LIN {X 0,Y 474.609,Z 227.864,A -85,B 0,C 180,E1 -7320.228,E2 -7320.228} C_VEL
LIN {X 0,Y 474.64,Z 227.86,A -85,B 0,C 180,E1 -7323.218,E2 -7323.218} C_VEL
LIN {X 0,Y 474.588,Z 227.869,A -85,B 0,C 180,E1 -7326.321,E2 -7326.321} C_VEL
LIN {X 0,Y 474.625,Z 227.862,A -85,B 0,C 180,E1 -7329.545,E2 -7329.545} C_VEL
LIN {X 0,Y 474.587,Z 227.87,A -85,B 0,C 180,E1 -7332.228,E2 -7332.228} C_VEL
LIN {X 0,Y 474.618,Z 227.86,A -85,B 0,C 180,E1 -7335.295,E2 -7335.295} C_VEL
LIN {X 0,Y 474.594,Z 227.868,A -85,B 0,C 180,E1 -7338.208,E2 -7338.208} C_VEL
LIN {X 0,Y 474.619,Z 227.864,A -85,B 0,C 180,E1 -7340.448,E2 -7340.448} C_VEL
LIN {X 0,Y 474.57,Z 227.865,A -85,B 0,C 180,E1 -7343.671,E2 -7343.671} C_VEL
LIN {X 0,Y 474.614,Z 227.864,A -85,B 0,C 180,E1 -7346.774,E2 -7346.774} C_VEL
LIN {X 0,Y 474.592,Z 227.863,A -85,B 0,C 180,E1 -7349.765,E2 -7349.765} C_VEL
LIN {X 0,Y 474.599,Z 227.867,A -85,B 0,C 180,E1 -7352.68,E2 -7352.68} C_VEL
LIN {X 0,Y 474.619,Z 227.86,A -85,B 0,C 180,E1 -7355.501,E2 -7355.501} C_VEL
LIN {X 0,Y 474.642,Z 227.86,A -85,B 0,C 180,E1 -7359.18,E2 -7359.18} C_VEL
LIN {X 0,Y 474.606,Z 227.861,A -85,B 0,C 180,E1 -7361.878,E2 -7361.878} C_VEL
LIN {X 0,Y 474.671,Z 227.856,A -85,B 0,C 180,E1 -7364.539,E2 -7364.539} C_VEL
LIN {X 0,Y 474.692,Z 227.848,A -85,B 0,C 180,E1 -7368.032,E2 -7368.032} C_VEL
LIN {X 0,Y 474.682,Z 227.855,A -85,B 0,C 180,E1 -7371.481,E2 -7371.481} C_VEL
LIN {X 0,Y 474.742,Z 227.843,A -85,B 0,C 180,E1 -7374.047,E2 -7374.047} C_VEL
LIN {X 0,Y 474.862,Z 227.835,A -85,B 0,C 180,E1 -7377.45,E2 -7377.45} C_VEL
LIN {X 0,Y 474.888,Z 227.826,A -85,B 0,C 180,E1 -7379.994,E2 -7379.994} C_VEL
LIN {X 0,Y 474.871,Z 227.828,A -85,B 0,C 180,E1 -7382.539,E2 -7382.539} C_VEL
LIN {X 0,Y 474.738,Z 227.848,A -85,B 0,C 180,E1 -7385.942,E2 -7385.942} C_VEL
LIN {X 0,Y 474.703,Z 227.851,A -85,B 0,C 180,E1 -7388.508,E2 -7388.508} C_VEL
LIN {X 0,Y 474.711,Z 227.853,A -85,B 0,C 180,E1 -7391.956,E2 -7391.956} C_VEL
LIN {X 0,Y 474.67,Z 227.86,A -85,B 0,C 180,E1 -7395.45,E2 -7395.45} C_VEL
LIN {X 0,Y 474.631,Z 227.862,A -85,B 0,C 180,E1 -7399.004,E2 -7399.004} C_VEL
LIN {X 0,Y 474.608,Z 227.868,A -85,B 0,C 180,E1 -7401.72,E2 -7401.72} C_VEL
LIN {X 0,Y 474.67,Z 227.981,A -85,B 0,C 180,E1 -7403.845,E2 -7403.845} C_VEL
LIN {X 0,Y 475.847,Z 234.41,A -85,B 0,C 180,E1 -7405.119,E2 -7405.119} C_VEL
LIN {X 0,Y 475.431,Z 251.659,A -85,B 0,C 180,E1 -7408.223,E2 -7408.223} C_VEL
LIN {X 0,Y 475.369,Z 257.615,A -85,B 0,C 180,E1 -7409.254,E2 -7409.254} C_VEL
LIN {X 0,Y 478.155,Z 273.903,A -85,B 0,C 180,E1 -7409.639,E2 -7409.639} C_VEL
LIN {X 0,Y 477.321,Z 365.648,A -85,B 0,C 180,E1 -7411.09,E2 -7411.09} C_VEL
LIN {X 0,Y 477,Z 379.548,A -85,B 0,C 180,E1 -7411.494,E2 -7411.494} C_VEL
LIN {X 0,Y 476.715,Z 392.201,A -85,B 0,C 180,E1 -7412.046,E2 -7412.046} C_VEL
LIN {X 0,Y 476.272,Z 404.083,A -85,B 0,C 180,E1 -7412.747,E2 -7412.747} C_VEL
LIN {X 0,Y 475.72,Z 415.798,A -85,B 0,C 180,E1 -7413.633,E2 -7413.633} C_VEL
LIN {X 0,Y 475.327,Z 425.567,A -85,B 0,C 180,E1 -7414.559,E2 -7414.559} C_VEL
LIN {X 0,Y 474.857,Z 435.029,A -85,B 0,C 180,E1 -7415.666,E2 -7415.666} C_VEL
LIN {X 0,Y 474.48,Z 443.518,A -85,B 0,C 180,E1 -7416.888,E2 -7416.888} C_VEL
LIN {X 0,Y 474.188,Z 451.047,A -85,B 0,C 180,E1 -7418.235,E2 -7418.235} C_VEL
LIN {X 0,Y 473.959,Z 457.052,A -85,B 0,C 180,E1 -7419.604,E2 -7419.604} C_VEL
LIN {X 0,Y 473.835,Z 461.346,A -85,B 0,C 180,E1 -7420.852,E2 -7420.852} C_VEL
LIN {X 0,Y 473.699,Z 464.658,A -85,B 0,C 180,E1 -7422.116,E2 -7422.116} C_VEL
LIN {X 0,Y 473.616,Z 466.97,A -85,B 0,C 180,E1 -7423.358,E2 -7423.358} C_VEL
LIN {X 0,Y 473.635,Z 468.364,A -85,B 0,C 180,E1 -7424.585,E2 -7424.585} C_VEL
LIN {X 0,Y 473.606,Z 468.909,A -85,B 0,C 180,E1 -7425.78,E2 -7425.78} C_VEL
LIN {X 0,Y 473.574,Z 468.694,A -85,B 0,C 180,E1 -7426.951,E2 -7426.951} C_VEL
LIN {X 0,Y 473.665,Z 467.748,A -85,B 0,C 180,E1 -7428.114,E2 -7428.114} C_VEL
LIN {X 0,Y 473.705,Z 464.944,A -85,B 0,C 180,E1 -7429.809,E2 -7429.809} C_VEL
LIN {X 0,Y 473.85,Z 460.634,A -85,B 0,C 180,E1 -7431.445,E2 -7431.445} C_VEL
LIN {X 0,Y 473.285,Z 458.514,A -85,B 0,C 180,E1 -7432.109,E2 -7432.109} C_VEL
LIN {X 0,Y 470.568,Z 454.555,A -85,B 0,C 180,E1 -7433.163,E2 -7433.163} C_VEL
LIN {X 0,Y 467.86,Z 449.885,A -85,B 0,C 180,E1 -7434.184,E2 -7434.184} C_VEL
LIN {X 0,Y 467.32,Z 446.646,A -85,B 0,C 180,E1 -7434.789,E2 -7434.789} C_VEL
LIN {X 0,Y 467.621,Z 439.191,A -85,B 0,C 180,E1 -7435.983,E2 -7435.983} C_VEL
LIN {X 0,Y 468.08,Z 429.769,A -85,B 0,C 180,E1 -7437.209,E2 -7437.209} C_VEL
LIN {X 0,Y 468.529,Z 420.264,A -85,B 0,C 180,E1 -7438.207,E2 -7438.207} C_VEL
LIN {X 0,Y 469.018,Z 409.141,A -85,B 0,C 180,E1 -7439.149,E2 -7439.149} C_VEL
LIN {X 0,Y 469.526,Z 397.344,A -85,B 0,C 180,E1 -7439.938,E2 -7439.938} C_VEL
LIN {X 0,Y 469.937,Z 385.154,A -85,B 0,C 180,E1 -7440.553,E2 -7440.553} C_VEL
LIN {X 0,Y 470.285,Z 372.084,A -85,B 0,C 180,E1 -7441.021,E2 -7441.021} C_VEL
LIN {X 0,Y 470.513,Z 359.082,A -85,B 0,C 180,E1 -7441.311,E2 -7441.311} C_VEL
LIN {X 0,Y 471.128,Z 273.425,A -85,B 0,C 180,E1 -7442.668,E2 -7442.668} C_VEL
LIN {X 0,Y 468.516,Z 258.548,A -85,B 0,C 180,E1 -7443.016,E2 -7443.016} C_VEL
LIN {X 0,Y 468.469,Z 257.54,A -85,B 0,C 180,E1 -7443.134,E2 -7443.134} C_VEL
LIN {X 0,Y 469.141,Z 241.607,A -85,B 0,C 180,E1 -7446.378,E2 -7446.378} C_VEL
LIN {X 0,Y 469.154,Z 237.141,A -85,B 0,C 180,E1 -7447.312,E2 -7447.312} C_VEL
LIN {X 0,Y 467.581,Z 228.795,A -85,B 0,C 180,E1 -7449.203,E2 -7449.203} C_VEL
LIN {X 0,Y 467.534,Z 228.751,A -85,B 0,C 180,E1 -7452.506,E2 -7452.506} C_VEL
LIN {X 0,Y 467.55,Z 228.741,A -85,B 0,C 180,E1 -7455.196,E2 -7455.196} C_VEL
LIN {X 0,Y 467.62,Z 228.731,A -85,B 0,C 180,E1 -7457.855,E2 -7457.855} C_VEL
LIN {X 0,Y 467.611,Z 228.733,A -85,B 0,C 180,E1 -7461.358,E2 -7461.358} C_VEL
LIN {X 0,Y 467.677,Z 228.724,A -85,B 0,C 180,E1 -7463.963,E2 -7463.963} C_VEL
LIN {X 0,Y 467.792,Z 228.712,A -85,B 0,C 180,E1 -7467.418,E2 -7467.418} C_VEL
LIN {X 0,Y 467.802,Z 228.708,A -85,B 0,C 180,E1 -7470.001,E2 -7470.001} C_VEL
LIN {X 0,Y 467.793,Z 228.711,A -85,B 0,C 180,E1 -7472.585,E2 -7472.585} C_VEL
LIN {X 0,Y 467.679,Z 228.724,A -85,B 0,C 180,E1 -7476.04,E2 -7476.04} C_VEL
LIN {X 0,Y 467.615,Z 228.732,A -85,B 0,C 180,E1 -7478.645,E2 -7478.645} C_VEL
LIN {X 0,Y 467.625,Z 228.731,A -85,B 0,C 180,E1 -7482.148,E2 -7482.148} C_VEL
LIN {X 0,Y 467.57,Z 228.744,A -85,B 0,C 180,E1 -7485.699,E2 -7485.699} C_VEL
LIN {X 0,Y 467.547,Z 228.74,A -85,B 0,C 180,E1 -7488.768,E2 -7488.768} C_VEL
LIN {X 0,Y 467.514,Z 228.747,A -85,B 0,C 180,E1 -7491.273,E2 -7491.273} C_VEL
LIN {X 0,Y 467.511,Z 228.751,A -85,B 0,C 180,E1 -7493.948,E2 -7493.948} C_VEL
LIN {X 0,Y 467.565,Z 228.738,A -85,B 0,C 180,E1 -7496.805,E2 -7496.805} C_VEL
LIN {X 0,Y 467.529,Z 228.747,A -85,B 0,C 180,E1 -7499.741,E2 -7499.741} C_VEL
LIN {X 0,Y 467.527,Z 228.743,A -85,B 0,C 180,E1 -7502.764,E2 -7502.764} C_VEL
LIN {X 0,Y 467.502,Z 228.75,A -85,B 0,C 180,E1 -7505.895,E2 -7505.895} C_VEL
LIN {X 0,Y 467.549,Z 228.74,A -85,B 0,C 180,E1 -7509.149,E2 -7509.149} C_VEL
LIN {X 0,Y 467.573,Z 228.744,A -85,B 0,C 180,E1 -7512.578,E2 -7512.578} C_VEL
LIN {X 0,Y 467.534,Z 228.746,A -85,B 0,C 180,E1 -7516.265,E2 -7516.265} C_VEL
LIN {X 0,Y 467.551,Z 228.747,A -85,B 0,C 180,E1 -7518.728,E2 -7518.728} C_VEL
LIN {X 0,Y 467.54,Z 228.742,A -85,B 0,C 180,E1 -7521.414,E2 -7521.414} C_VEL
LIN {X 0,Y 467.529,Z 228.744,A -85,B 0,C 180,E1 -7524.268,E2 -7524.268} C_VEL
LIN {X 0,Y 467.551,Z 228.743,A -85,B 0,C 180,E1 -7527.328,E2 -7527.328} C_VEL
LIN {X 0,Y 467.544,Z 228.744,A -85,B 0,C 180,E1 -7530.675,E2 -7530.675} C_VEL
LIN {X 0,Y 467.594,Z 228.742,A -85,B 0,C 180,E1 -7533.207,E2 -7533.207} C_VEL
LIN {X 0,Y 467.574,Z 228.737,A -85,B 0,C 180,E1 -7536.475,E2 -7536.475} C_VEL
LIN {X 0,Y 467.608,Z 228.735,A -85,B 0,C 180,E1 -7539.784,E2 -7539.784} C_VEL
LIN {X 0,Y 467.586,Z 228.735,A -85,B 0,C 180,E1 -7542.513,E2 -7542.513} C_VEL
LIN {X 0,Y 467.596,Z 228.737,A -85,B 0,C 180,E1 -7545.203,E2 -7545.203} C_VEL
LIN {X 0,Y 467.65,Z 228.733,A -85,B 0,C 180,E1 -7547.861,E2 -7547.861} C_VEL
LIN {X 0,Y 467.667,Z 228.728,A -85,B 0,C 180,E1 -7551.363,E2 -7551.363} C_VEL
LIN {X 0,Y 467.712,Z 228.727,A -85,B 0,C 180,E1 -7553.968,E2 -7553.968} C_VEL
LIN {X 0,Y 467.851,Z 228.704,A -85,B 0,C 180,E1 -7557.423,E2 -7557.423} C_VEL
LIN {X 0,Y 467.854,Z 228.71,A -85,B 0,C 180,E1 -7560.006,E2 -7560.006} C_VEL
LIN {X 0,Y 467.819,Z 228.709,A -85,B 0,C 180,E1 -7562.589,E2 -7562.589} C_VEL
LIN {X 0,Y 467.714,Z 228.725,A -85,B 0,C 180,E1 -7566.043,E2 -7566.043} C_VEL
LIN {X 0,Y 467.646,Z 228.732,A -85,B 0,C 180,E1 -7568.649,E2 -7568.649} C_VEL
LIN {X 0,Y 467.669,Z 228.729,A -85,B 0,C 180,E1 -7572.15,E2 -7572.15} C_VEL
LIN {X 0,Y 467.664,Z 228.726,A -85,B 0,C 180,E1 -7575.889,E2 -7575.889} C_VEL
LIN {X 0,Y 467.636,Z 228.73,A -85,B 0,C 180,E1 -7579.312,E2 -7579.312} C_VEL
LIN {X 0,Y 467.548,Z 228.74,A -85,B 0,C 180,E1 -7582.078,E2 -7582.078} C_VEL
LIN {X 0,Y 467.574,Z 228.746,A -85,B 0,C 180,E1 -7584.893,E2 -7584.893} C_VEL
LIN {X 0,Y 467.564,Z 228.738,A -85,B 0,C 180,E1 -7587.777,E2 -7587.777} C_VEL
LIN {X 0,Y 467.566,Z 228.745,A -85,B 0,C 180,E1 -7591.043,E2 -7591.043} C_VEL
LIN {X 0,Y 467.595,Z 228.734,A -85,B 0,C 180,E1 -7594.242,E2 -7594.242} C_VEL
LIN {X 0,Y 467.561,Z 228.745,A -85,B 0,C 180,E1 -7597.187,E2 -7597.187} C_VEL
LIN {X 0,Y 467.577,Z 228.736,A -85,B 0,C 180,E1 -7600.269,E2 -7600.269} C_VEL
LIN {X 0,Y 467.537,Z 228.741,A -85,B 0,C 180,E1 -7602.57,E2 -7602.57} C_VEL
LIN {X 0,Y 467.574,Z 228.738,A -85,B 0,C 180,E1 -7605.052,E2 -7605.052} C_VEL
LIN {X 0,Y 467.58,Z 228.736,A -85,B 0,C 180,E1 -7608.727,E2 -7608.727} C_VEL
LIN {X 0,Y 467.562,Z 228.745,A -85,B 0,C 180,E1 -7611.954,E2 -7611.954} C_VEL
LIN {X 0,Y 467.573,Z 228.737,A -85,B 0,C 180,E1 -7615.167,E2 -7615.167} C_VEL
LIN {X 0,Y 467.596,Z 228.742,A -85,B 0,C 180,E1 -7618.26,E2 -7618.26} C_VEL
LIN {X 0,Y 467.573,Z 228.74,A -85,B 0,C 180,E1 -7621.249,E2 -7621.249} C_VEL
LIN {X 0,Y 467.6,Z 228.742,A -85,B 0,C 180,E1 -7624.158,E2 -7624.158} C_VEL
LIN {X 0,Y 467.637,Z 228.864,A -85,B 0,C 180,E1 -7625.061,E2 -7625.061} C_VEL
LIN {X 0,Y 469.628,Z 239.857,A -85,B 0,C 180,E1 -7627.333,E2 -7627.333} C_VEL
LIN {X 0,Y 469.11,Z 253.106,A -85,B 0,C 180,E1 -7629.843,E2 -7629.843} C_VEL
LIN {X 0,Y 468.404,Z 270.161,A -85,B 0,C 180,E1 -7632.986,E2 -7632.986} C_VEL
LIN {X 0,Y 469.313,Z 275.962,A -85,B 0,C 180,E1 -7633.15,E2 -7633.15} C_VEL
LIN {X 0,Y 471.214,Z 288.215,A -85,B 0,C 180,E1 -7633.414,E2 -7633.414} C_VEL
LIN {X 0,Y 470.431,Z 377.814,A -85,B 0,C 180,E1 -7634.843,E2 -7634.843} C_VEL
LIN {X 0,Y 470.097,Z 391.028,A -85,B 0,C 180,E1 -7635.22,E2 -7635.22} C_VEL
LIN {X 0,Y 469.668,Z 403.753,A -85,B 0,C 180,E1 -7635.76,E2 -7635.76} C_VEL
LIN {X 0,Y 469.197,Z 415.879,A -85,B 0,C 180,E1 -7636.463,E2 -7636.463} C_VEL
LIN {X 0,Y 468.757,Z 426.287,A -85,B 0,C 180,E1 -7637.236,E2 -7637.236} C_VEL
LIN {X 0,Y 468.268,Z 436.753,A -85,B 0,C 180,E1 -7638.199,E2 -7638.199} C_VEL
LIN {X 0,Y 467.808,Z 445.435,A -85,B 0,C 180,E1 -7639.175,E2 -7639.175} C_VEL
LIN {X 0,Y 467.479,Z 453.433,A -85,B 0,C 180,E1 -7640.261,E2 -7640.261} C_VEL
LIN {X 0,Y 467.157,Z 461.253,A -85,B 0,C 180,E1 -7641.564,E2 -7641.564} C_VEL
LIN {X 0,Y 466.862,Z 468.418,A -85,B 0,C 180,E1 -7643.082,E2 -7643.082} C_VEL
LIN {X 0,Y 466.795,Z 473.191,A -85,B 0,C 180,E1 -7644.382,E2 -7644.382} C_VEL
LIN {X 0,Y 466.651,Z 476.837,A -85,B 0,C 180,E1 -7645.68,E2 -7645.68} C_VEL
LIN {X 0,Y 466.665,Z 478.72,A -85,B 0,C 180,E1 -7646.545,E2 -7646.545} C_VEL
LIN {X 0,Y 466.648,Z 480.133,A -85,B 0,C 180,E1 -7647.409,E2 -7647.409} C_VEL
LIN {X 0,Y 466.593,Z 481.751,A -85,B 0,C 180,E1 -7649.135,E2 -7649.135} C_VEL
LIN {X 0,Y 466.603,Z 481.973,A -85,B 0,C 180,E1 -7649.999,E2 -7649.999} C_VEL
LIN {X 0,Y 466.593,Z 481.757,A -85,B 0,C 180,E1 -7650.862,E2 -7650.862} C_VEL
LIN {X 0,Y 466.648,Z 480.142,A -85,B 0,C 180,E1 -7652.588,E2 -7652.588} C_VEL
LIN {X 0,Y 466.664,Z 478.736,A -85,B 0,C 180,E1 -7653.452,E2 -7653.452} C_VEL
LIN {X 0,Y 466.694,Z 475.781,A -85,B 0,C 180,E1 -7654.749,E2 -7654.749} C_VEL
LIN {X 0,Y 466.779,Z 471.78,A -85,B 0,C 180,E1 -7656.048,E2 -7656.048} C_VEL
LIN {X 0,Y 466.983,Z 465.623,A -85,B 0,C 180,E1 -7657.565,E2 -7657.565} C_VEL
LIN {X 0,Y 467.274,Z 458.899,A -85,B 0,C 180,E1 -7658.867,E2 -7658.867} C_VEL
LIN {X 0,Y 467.616,Z 450.554,A -85,B 0,C 180,E1 -7660.17,E2 -7660.17} C_VEL
LIN {X 0,Y 468.03,Z 441.975,A -85,B 0,C 180,E1 -7661.255,E2 -7661.255} C_VEL
LIN {X 0,Y 468.555,Z 431.775,A -85,B 0,C 180,E1 -7662.304,E2 -7662.304} C_VEL
LIN {X 0,Y 468.977,Z 420.901,A -85,B 0,C 180,E1 -7663.209,E2 -7663.209} C_VEL
LIN {X 0,Y 469.468,Z 409.359,A -85,B 0,C 180,E1 -7663.967,E2 -7663.967} C_VEL
LIN {X 0,Y 469.935,Z 397.4,A -85,B 0,C 180,E1 -7664.561,E2 -7664.561} C_VEL
LIN {X 0,Y 470.353,Z 383.614,A -85,B 0,C 180,E1 -7665.046,E2 -7665.046} C_VEL
LIN {X 0,Y 470.587,Z 370.995,A -85,B 0,C 180,E1 -7665.315,E2 -7665.315} C_VEL
LIN {X 0,Y 471.217,Z 286.858,A -85,B 0,C 180,E1 -7666.654,E2 -7666.654} C_VEL
LIN {X 0,Y 468.38,Z 269.763,A -85,B 0,C 180,E1 -7667.072,E2 -7667.072} C_VEL
LIN {X 0,Y 468.952,Z 253.914,A -85,B 0,C 180,E1 -7669.933,E2 -7669.933} C_VEL
LIN {X 0,Y 469.534,Z 240.329,A -85,B 0,C 180,E1 -7672.436,E2 -7672.436} C_VEL
LIN {X 0,Y 468.428,Z 232.889,A -85,B 0,C 180,E1 -7673.895,E2 -7673.895} C_VEL
LIN {X 0,Y 467.616,Z 228.82,A -85,B 0,C 180,E1 -7674.766,E2 -7674.766} C_VEL
LIN {X 0,Y 467.623,Z 228.738,A -85,B 0,C 180,E1 -7677.767,E2 -7677.767} C_VEL
LIN {X 0,Y 467.573,Z 228.738,A -85,B 0,C 180,E1 -7681.041,E2 -7681.041} C_VEL
LIN {X 0,Y 467.594,Z 228.74,A -85,B 0,C 180,E1 -7684.239,E2 -7684.239} C_VEL
LIN {X 0,Y 467.546,Z 228.743,A -85,B 0,C 180,E1 -7687.182,E2 -7687.182} C_VEL
LIN {X 0,Y 467.562,Z 228.745,A -85,B 0,C 180,E1 -7690.264,E2 -7690.264} C_VEL
LIN {X 0,Y 467.549,Z 228.743,A -85,B 0,C 180,E1 -7693.742,E2 -7693.742} C_VEL
LIN {X 0,Y 467.547,Z 228.748,A -85,B 0,C 180,E1 -7696.251,E2 -7696.251} C_VEL
LIN {X 0,Y 467.558,Z 228.742,A -85,B 0,C 180,E1 -7699.729,E2 -7699.729} C_VEL
LIN {X 0,Y 467.516,Z 228.746,A -85,B 0,C 180,E1 -7702.815,E2 -7702.815} C_VEL
LIN {X 0,Y 467.575,Z 228.739,A -85,B 0,C 180,E1 -7705.756,E2 -7705.756} C_VEL
LIN {X 0,Y 467.545,Z 228.743,A -85,B 0,C 180,E1 -7708.956,E2 -7708.956} C_VEL
LIN {X 0,Y 467.541,Z 228.746,A -85,B 0,C 180,E1 -7712.222,E2 -7712.222} C_VEL
LIN {X 0,Y 467.551,Z 228.744,A -85,B 0,C 180,E1 -7715.105,E2 -7715.105} C_VEL
LIN {X 0,Y 467.517,Z 228.743,A -85,B 0,C 180,E1 -7717.921,E2 -7717.921} C_VEL
LIN {X 0,Y 467.546,Z 228.745,A -85,B 0,C 180,E1 -7720.684,E2 -7720.684} C_VEL
LIN {X 0,Y 467.585,Z 228.735,A -85,B 0,C 180,E1 -7724.135,E2 -7724.135} C_VEL
LIN {X 0,Y 467.643,Z 228.727,A -85,B 0,C 180,E1 -7727.638,E2 -7727.638} C_VEL
LIN {X 0,Y 467.642,Z 228.733,A -85,B 0,C 180,E1 -7731.351,E2 -7731.351} C_VEL
LIN {X 0,Y 467.707,Z 228.719,A -85,B 0,C 180,E1 -7733.957,E2 -7733.957} C_VEL
LIN {X 0,Y 467.803,Z 228.714,A -85,B 0,C 180,E1 -7737.411,E2 -7737.411} C_VEL
LIN {X 0,Y 467.859,Z 228.701,A -85,B 0,C 180,E1 -7739.994,E2 -7739.994} C_VEL
LIN {X 0,Y 467.837,Z 228.705,A -85,B 0,C 180,E1 -7742.577,E2 -7742.577} C_VEL
LIN {X 0,Y 467.7,Z 228.724,A -85,B 0,C 180,E1 -7746.032,E2 -7746.032} C_VEL
LIN {X 0,Y 467.657,Z 228.729,A -85,B 0,C 180,E1 -7748.637,E2 -7748.637} C_VEL
LIN {X 0,Y 467.663,Z 228.728,A -85,B 0,C 180,E1 -7752.373,E2 -7752.373} C_VEL
LIN {X 0,Y 467.618,Z 228.739,A -85,B 0,C 180,E1 -7755.88,E2 -7755.88} C_VEL
LIN {X 0,Y 467.59,Z 228.741,A -85,B 0,C 180,E1 -7759.302,E2 -7759.302} C_VEL
LIN {X 0,Y 467.543,Z 228.748,A -85,B 0,C 180,E1 -7762.066,E2 -7762.066} C_VEL
LIN {X 0,Y 467.633,Z 228.785,A -85,B 0,C 180,E1 -7763.61,E2 -7763.61} C_VEL
LIN {X 0,Y 468.567,Z 233.439,A -85,B 0,C 180,E1 -7764.588,E2 -7764.588} C_VEL
LIN {X 0,Y 468.961,Z 237.071,A -85,B 0,C 180,E1 -7765.276,E2 -7765.276} C_VEL
LIN {X 0,Y 468.449,Z 254.311,A -85,B 0,C 180,E1 -7768.413,E2 -7768.413} C_VEL
LIN {X 0,Y 468.408,Z 257.7,A -85,B 0,C 180,E1 -7768.985,E2 -7768.985} C_VEL
LIN {X 0,Y 471.352,Z 273.713,A -85,B 0,C 180,E1 -7769.382,E2 -7769.382} C_VEL
LIN {X 0,Y 470.48,Z 366.047,A -85,B 0,C 180,E1 -7770.872,E2 -7770.872} C_VEL
LIN {X 0,Y 470.127,Z 380.038,A -85,B 0,C 180,E1 -7771.289,E2 -7771.289} C_VEL
LIN {X 0,Y 469.829,Z 391.909,A -85,B 0,C 180,E1 -7771.813,E2 -7771.813} C_VEL
LIN {X 0,Y 469.359,Z 403.284,A -85,B 0,C 180,E1 -7772.482,E2 -7772.482} C_VEL
LIN {X 0,Y 468.822,Z 415.254,A -85,B 0,C 180,E1 -7773.39,E2 -7773.39} C_VEL
LIN {X 0,Y 468.349,Z 425.658,A -85,B 0,C 180,E1 -7774.382,E2 -7774.382} C_VEL
LIN {X 0,Y 467.838,Z 435.416,A -85,B 0,C 180,E1 -7775.544,E2 -7775.544} C_VEL
LIN {X 0,Y 467.468,Z 443.261,A -85,B 0,C 180,E1 -7776.689,E2 -7776.689} C_VEL
LIN {X 0,Y 467.138,Z 450.965,A -85,B 0,C 180,E1 -7778.075,E2 -7778.075} C_VEL
LIN {X 0,Y 466.883,Z 457.229,A -85,B 0,C 180,E1 -7779.523,E2 -7779.523} C_VEL
LIN {X 0,Y 466.728,Z 462.57,A -85,B 0,C 180,E1 -7781.161,E2 -7781.161} C_VEL
LIN {X 0,Y 466.579,Z 465.989,A -85,B 0,C 180,E1 -7782.663,E2 -7782.663} C_VEL
LIN {X 0,Y 466.535,Z 467.769,A -85,B 0,C 180,E1 -7783.853,E2 -7783.853} C_VEL
LIN {X 0,Y 466.532,Z 468.774,A -85,B 0,C 180,E1 -7785.062,E2 -7785.062} C_VEL
LIN {X 0,Y 466.475,Z 469.004,A -85,B 0,C 180,E1 -7786.305,E2 -7786.305} C_VEL
LIN {X 0,Y 466.508,Z 468.399,A -85,B 0,C 180,E1 -7787.565,E2 -7787.565} C_VEL
LIN {X 0,Y 466.569,Z 466.896,A -85,B 0,C 180,E1 -7788.851,E2 -7788.851} C_VEL
LIN {X 0,Y 466.628,Z 464.383,A -85,B 0,C 180,E1 -7790.172,E2 -7790.172} C_VEL
LIN {X 0,Y 466.774,Z 460.754,A -85,B 0,C 180,E1 -7791.516,E2 -7791.516} C_VEL
LIN {X 0,Y 466.963,Z 455.403,A -85,B 0,C 180,E1 -7792.988,E2 -7792.988} C_VEL
LIN {X 0,Y 467.205,Z 449.264,A -85,B 0,C 180,E1 -7794.306,E2 -7794.306} C_VEL
LIN {X 0,Y 467.32,Z 446.646,A -85,B 0,C 180,E1 -7794.789,E2 -7794.789} C_VEL
LIN {X 0,Y 466.807,Z 443.26,A -85,B 0,C 180,E1 -7795.377,E2 -7795.377} C_VEL
LIN {X 0,Y 464.234,Z 437.436,A -85,B 0,C 180,E1 -7796.313,E2 -7796.313} C_VEL
LIN {X 0,Y 461.697,Z 431.084,A -85,B 0,C 180,E1 -7797.202,E2 -7797.202} C_VEL
LIN {X 0,Y 461.245,Z 426.806,A -85,B 0,C 180,E1 -7797.712,E2 -7797.712} C_VEL
LIN {X 0,Y 461.776,Z 416.304,A -85,B 0,C 180,E1 -7798.755,E2 -7798.755} C_VEL
LIN {X 0,Y 462.293,Z 405.076,A -85,B 0,C 180,E1 -7799.639,E2 -7799.639} C_VEL
LIN {X 0,Y 462.766,Z 393.347,A -85,B 0,C 180,E1 -7800.364,E2 -7800.364} C_VEL
LIN {X 0,Y 463.168,Z 380.581,A -85,B 0,C 180,E1 -7800.953,E2 -7800.953} C_VEL
LIN {X 0,Y 463.522,Z 367.51,A -85,B 0,C 180,E1 -7801.358,E2 -7801.358} C_VEL
LIN {X 0,Y 463.75,Z 344.948,A -85,B 0,C 180,E1 -7801.755,E2 -7801.755} C_VEL
LIN {X 0,Y 464.275,Z 273.94,A -85,B 0,C 180,E1 -7802.902,E2 -7802.902} C_VEL
LIN {X 0,Y 461.546,Z 258.523,A -85,B 0,C 180,E1 -7803.279,E2 -7803.279} C_VEL
LIN {X 0,Y 461.528,Z 256.772,A -85,B 0,C 180,E1 -7803.553,E2 -7803.553} C_VEL
LIN {X 0,Y 462.19,Z 242.567,A -85,B 0,C 180,E1 -7806.502,E2 -7806.502} C_VEL
LIN {X 0,Y 462.17,Z 238.23,A -85,B 0,C 180,E1 -7807.422,E2 -7807.422} C_VEL
LIN {X 0,Y 460.515,Z 229.675,A -85,B 0,C 180,E1 -7809.395,E2 -7809.395} C_VEL
LIN {X 0,Y 460.483,Z 229.627,A -85,B 0,C 180,E1 -7812.229,E2 -7812.229} C_VEL
LIN {X 0,Y 460.51,Z 229.62,A -85,B 0,C 180,E1 -7814.965,E2 -7814.965} C_VEL
LIN {X 0,Y 460.6,Z 229.605,A -85,B 0,C 180,E1 -7817.667,E2 -7817.667} C_VEL
LIN {X 0,Y 460.558,Z 229.613,A -85,B 0,C 180,E1 -7821.224,E2 -7821.224} C_VEL
LIN {X 0,Y 460.641,Z 229.6,A -85,B 0,C 180,E1 -7823.871,E2 -7823.871} C_VEL
LIN {X 0,Y 460.758,Z 229.588,A -85,B 0,C 180,E1 -7827.379,E2 -7827.379} C_VEL
LIN {X 0,Y 460.774,Z 229.583,A -85,B 0,C 180,E1 -7830.001,E2 -7830.001} C_VEL
LIN {X 0,Y 460.759,Z 229.588,A -85,B 0,C 180,E1 -7832.624,E2 -7832.624} C_VEL
LIN {X 0,Y 460.643,Z 229.6,A -85,B 0,C 180,E1 -7836.132,E2 -7836.132} C_VEL
LIN {X 0,Y 460.561,Z 229.612,A -85,B 0,C 180,E1 -7838.779,E2 -7838.779} C_VEL
LIN {X 0,Y 460.562,Z 229.61,A -85,B 0,C 180,E1 -7842.46,E2 -7842.46} C_VEL
LIN {X 0,Y 460.53,Z 229.617,A -85,B 0,C 180,E1 -7846.001,E2 -7846.001} C_VEL
LIN {X 0,Y 460.501,Z 229.618,A -85,B 0,C 180,E1 -7848.905,E2 -7848.905} C_VEL
LIN {X 0,Y 460.449,Z 229.629,A -85,B 0,C 180,E1 -7851.49,E2 -7851.49} C_VEL
LIN {X 0,Y 460.483,Z 229.622,A -85,B 0,C 180,E1 -7854.337,E2 -7854.337} C_VEL
LIN {X 0,Y 460.522,Z 229.616,A -85,B 0,C 180,E1 -7857.248,E2 -7857.248} C_VEL
LIN {X 0,Y 460.47,Z 229.627,A -85,B 0,C 180,E1 -7860.244,E2 -7860.244} C_VEL
LIN {X 0,Y 460.473,Z 229.621,A -85,B 0,C 180,E1 -7863.331,E2 -7863.331} C_VEL
LIN {X 0,Y 460.425,Z 229.632,A -85,B 0,C 180,E1 -7866.535,E2 -7866.535} C_VEL
LIN {X 0,Y 460.525,Z 229.617,A -85,B 0,C 180,E1 -7869.864,E2 -7869.864} C_VEL
LIN {X 0,Y 460.496,Z 229.621,A -85,B 0,C 180,E1 -7872.911,E2 -7872.911} C_VEL
LIN {X 0,Y 460.481,Z 229.621,A -85,B 0,C 180,E1 -7875.836,E2 -7875.836} C_VEL
LIN {X 0,Y 460.505,Z 229.621,A -85,B 0,C 180,E1 -7878.997,E2 -7878.997} C_VEL
LIN {X 0,Y 460.509,Z 229.619,A -85,B 0,C 180,E1 -7881.276,E2 -7881.276} C_VEL
LIN {X 0,Y 460.479,Z 229.625,A -85,B 0,C 180,E1 -7884.562,E2 -7884.562} C_VEL
LIN {X 0,Y 460.502,Z 229.618,A -85,B 0,C 180,E1 -7887.723,E2 -7887.723} C_VEL
LIN {X 0,Y 460.514,Z 229.62,A -85,B 0,C 180,E1 -7890.776,E2 -7890.776} C_VEL
LIN {X 0,Y 460.538,Z 229.615,A -85,B 0,C 180,E1 -7893.742,E2 -7893.742} C_VEL
LIN {X 0,Y 460.528,Z 229.615,A -85,B 0,C 180,E1 -7896.631,E2 -7896.631} C_VEL
LIN {X 0,Y 460.537,Z 229.621,A -85,B 0,C 180,E1 -7899.46,E2 -7899.46} C_VEL
LIN {X 0,Y 460.537,Z 229.613,A -85,B 0,C 180,E1 -7902.237,E2 -7902.237} C_VEL
LIN {X 0,Y 460.555,Z 229.612,A -85,B 0,C 180,E1 -7904.972,E2 -7904.972} C_VEL
LIN {X 0,Y 460.604,Z 229.605,A -85,B 0,C 180,E1 -7908.566,E2 -7908.566} C_VEL
LIN {X 0,Y 460.617,Z 229.605,A -85,B 0,C 180,E1 -7911.23,E2 -7911.23} C_VEL
LIN {X 0,Y 460.678,Z 229.604,A -85,B 0,C 180,E1 -7913.876,E2 -7913.876} C_VEL
LIN {X 0,Y 460.791,Z 229.583,A -85,B 0,C 180,E1 -7917.383,E2 -7917.383} C_VEL
LIN {X 0,Y 460.823,Z 229.586,A -85,B 0,C 180,E1 -7920.006,E2 -7920.006} C_VEL
LIN {X 0,Y 460.763,Z 229.587,A -85,B 0,C 180,E1 -7922.628,E2 -7922.628} C_VEL
LIN {X 0,Y 460.679,Z 229.602,A -85,B 0,C 180,E1 -7926.136,E2 -7926.136} C_VEL
LIN {X 0,Y 460.602,Z 229.608,A -85,B 0,C 180,E1 -7928.782,E2 -7928.782} C_VEL
LIN {X 0,Y 460.623,Z 229.609,A -85,B 0,C 180,E1 -7932.339,E2 -7932.339} C_VEL
LIN {X 0,Y 460.617,Z 229.604,A -85,B 0,C 180,E1 -7936.002,E2 -7936.002} C_VEL
LIN {X 0,Y 460.582,Z 229.607,A -85,B 0,C 180,E1 -7939.62,E2 -7939.62} C_VEL
LIN {X 0,Y 460.525,Z 229.618,A -85,B 0,C 180,E1 -7942.433,E2 -7942.433} C_VEL
LIN {X 0,Y 460.551,Z 229.611,A -85,B 0,C 180,E1 -7945.796,E2 -7945.796} C_VEL
LIN {X 0,Y 460.539,Z 229.619,A -85,B 0,C 180,E1 -7949.235,E2 -7949.235} C_VEL
LIN {X 0,Y 460.537,Z 229.613,A -85,B 0,C 180,E1 -7952.288,E2 -7952.288} C_VEL
LIN {X 0,Y 460.524,Z 229.621,A -85,B 0,C 180,E1 -7955.449,E2 -7955.449} C_VEL
LIN {X 0,Y 460.523,Z 229.617,A -85,B 0,C 180,E1 -7958.893,E2 -7958.893} C_VEL
LIN {X 0,Y 460.522,Z 229.622,A -85,B 0,C 180,E1 -7961.6,E2 -7961.6} C_VEL
LIN {X 0,Y 460.517,Z 229.615,A -85,B 0,C 180,E1 -7964.593,E2 -7964.593} C_VEL
LIN {X 0,Y 460.493,Z 229.626,A -85,B 0,C 180,E1 -7967.814,E2 -7967.814} C_VEL
LIN {X 0,Y 460.529,Z 229.618,A -85,B 0,C 180,E1 -7970.136,E2 -7970.136} C_VEL
LIN {X 0,Y 460.484,Z 229.623,A -85,B 0,C 180,E1 -7973.47,E2 -7973.47} C_VEL
LIN {X 0,Y 460.535,Z 229.614,A -85,B 0,C 180,E1 -7976.674,E2 -7976.674} C_VEL
LIN {X 0,Y 460.524,Z 229.619,A -85,B 0,C 180,E1 -7979.76,E2 -7979.76} C_VEL
LIN {X 0,Y 460.552,Z 229.618,A -85,B 0,C 180,E1 -7982.754,E2 -7982.754} C_VEL
LIN {X 0,Y 460.572,Z 229.687,A -85,B 0,C 180,E1 -7984.826,E2 -7984.826} C_VEL
LIN {X 0,Y 461.616,Z 235.024,A -85,B 0,C 180,E1 -7985.997,E2 -7985.997} C_VEL
LIN {X 0,Y 462.707,Z 242.134,A -85,B 0,C 180,E1 -7987.447,E2 -7987.447} C_VEL
LIN {X 0,Y 461.887,Z 258.794,A -85,B 0,C 180,E1 -7990.633,E2 -7990.633} C_VEL
LIN {X 0,Y 461.455,Z 270.242,A -85,B 0,C 180,E1 -7992.747,E2 -7992.747} C_VEL
LIN {X 0,Y 464.377,Z 288.238,A -85,B 0,C 180,E1 -7993.173,E2 -7993.173} C_VEL
LIN {X 0,Y 463.554,Z 378.276,A -85,B 0,C 180,E1 -7994.641,E2 -7994.641} C_VEL
LIN {X 0,Y 463.174,Z 392.057,A -85,B 0,C 180,E1 -7995.05,E2 -7995.05} C_VEL
LIN {X 0,Y 462.737,Z 404.472,A -85,B 0,C 180,E1 -7995.598,E2 -7995.598} C_VEL
LIN {X 0,Y 462.262,Z 415.574,A -85,B 0,C 180,E1 -7996.256,E2 -7996.256} C_VEL
LIN {X 0,Y 461.761,Z 426.972,A -85,B 0,C 180,E1 -7997.121,E2 -7997.121} C_VEL
LIN {X 0,Y 461.241,Z 437.593,A -85,B 0,C 180,E1 -7998.128,E2 -7998.128} C_VEL
LIN {X 0,Y 460.742,Z 446.968,A -85,B 0,C 180,E1 -7999.229,E2 -7999.229} C_VEL
LIN {X 0,Y 460.296,Z 456.035,A -85,B 0,C 180,E1 -8000.552,E2 -8000.552} C_VEL
LIN {X 0,Y 460.016,Z 463.339,A -85,B 0,C 180,E1 -8001.874,E2 -8001.874} C_VEL
LIN {X 0,Y 459.758,Z 469.467,A -85,B 0,C 180,E1 -8003.271,E2 -8003.271} C_VEL
LIN {X 0,Y 459.687,Z 474.395,A -85,B 0,C 180,E1 -8004.735,E2 -8004.735} C_VEL
LIN {X 0,Y 459.569,Z 476.714,A -85,B 0,C 180,E1 -8005.613,E2 -8005.613} C_VEL
LIN {X 0,Y 459.562,Z 478.604,A -85,B 0,C 180,E1 -8006.492,E2 -8006.492} C_VEL
LIN {X 0,Y 459.571,Z 480.024,A -85,B 0,C 180,E1 -8007.369,E2 -8007.369} C_VEL
LIN {X 0,Y 459.499,Z 481.649,A -85,B 0,C 180,E1 -8009.122,E2 -8009.122} C_VEL
LIN {X 0,Y 459.505,Z 481.874,A -85,B 0,C 180,E1 -8009.999,E2 -8009.999} C_VEL
LIN {X 0,Y 459.499,Z 481.662,A -85,B 0,C 180,E1 -8010.875,E2 -8010.875} C_VEL
LIN {X 0,Y 459.571,Z 480.052,A -85,B 0,C 180,E1 -8012.628,E2 -8012.628} C_VEL
LIN {X 0,Y 459.561,Z 478.647,A -85,B 0,C 180,E1 -8013.506,E2 -8013.506} C_VEL
LIN {X 0,Y 459.626,Z 475.694,A -85,B 0,C 180,E1 -8014.823,E2 -8014.823} C_VEL
LIN {X 0,Y 459.725,Z 470.655,A -85,B 0,C 180,E1 -8016.429,E2 -8016.429} C_VEL
LIN {X 0,Y 459.955,Z 464.522,A -85,B 0,C 180,E1 -8017.903,E2 -8017.903} C_VEL
LIN {X 0,Y 460.241,Z 457.57,A -85,B 0,C 180,E1 -8019.225,E2 -8019.225} C_VEL
LIN {X 0,Y 460.643,Z 448.858,A -85,B 0,C 180,E1 -8020.548,E2 -8020.548} C_VEL
LIN {X 0,Y 461.197,Z 439.93,A -85,B 0,C 180,E1 -8021.647,E2 -8021.647} C_VEL
LIN {X 0,Y 461.729,Z 430.057,A -85,B 0,C 180,E1 -8022.643,E2 -8022.643} C_VEL
LIN {X 0,Y 462.128,Z 419.367,A -85,B 0,C 180,E1 -8023.52,E2 -8023.52} C_VEL
LIN {X 0,Y 462.656,Z 407.301,A -85,B 0,C 180,E1 -8024.289,E2 -8024.289} C_VEL
LIN {X 0,Y 463.14,Z 396.043,A -85,B 0,C 180,E1 -8024.835,E2 -8024.835} C_VEL
LIN {X 0,Y 463.546,Z 382.644,A -85,B 0,C 180,E1 -8025.3,E2 -8025.3} C_VEL
LIN {X 0,Y 463.851,Z 367.633,A -85,B 0,C 180,E1 -8025.599,E2 -8025.599} C_VEL
LIN {X 0,Y 464.4,Z 287.53,A -85,B 0,C 180,E1 -8026.904,E2 -8026.904} C_VEL
LIN {X 0,Y 461.434,Z 269.693,A -85,B 0,C 180,E1 -8027.347,E2 -8027.347} C_VEL
LIN {X 0,Y 462.086,Z 253.855,A -85,B 0,C 180,E1 -8030.242,E2 -8030.242} C_VEL
LIN {X 0,Y 462.614,Z 241.506,A -85,B 0,C 180,E1 -8032.555,E2 -8032.555} C_VEL
LIN {X 0,Y 461.511,Z 234.384,A -85,B 0,C 180,E1 -8033.974,E2 -8033.974} C_VEL
LIN {X 0,Y 460.579,Z 229.692,A -85,B 0,C 180,E1 -8034.99,E2 -8034.99} C_VEL
LIN {X 0,Y 460.556,Z 229.617,A -85,B 0,C 180,E1 -8038.231,E2 -8038.231} C_VEL
LIN {X 0,Y 460.528,Z 229.617,A -85,B 0,C 180,E1 -8041.28,E2 -8041.28} C_VEL
LIN {X 0,Y 460.536,Z 229.618,A -85,B 0,C 180,E1 -8044.502,E2 -8044.502} C_VEL
LIN {X 0,Y 460.503,Z 229.624,A -85,B 0,C 180,E1 -8047.62,E2 -8047.62} C_VEL
LIN {X 0,Y 460.52,Z 229.616,A -85,B 0,C 180,E1 -8051.01,E2 -8051.01} C_VEL
LIN {X 0,Y 460.514,Z 229.62,A -85,B 0,C 180,E1 -8054.586,E2 -8054.586} C_VEL
LIN {X 0,Y 460.477,Z 229.625,A -85,B 0,C 180,E1 -8057.809,E2 -8057.809} C_VEL
LIN {X 0,Y 460.511,Z 229.624,A -85,B 0,C 180,E1 -8060.131,E2 -8060.131} C_VEL
LIN {X 0,Y 460.459,Z 229.622,A -85,B 0,C 180,E1 -8063.465,E2 -8063.465} C_VEL
LIN {X 0,Y 460.516,Z 229.62,A -85,B 0,C 180,E1 -8066.67,E2 -8066.67} C_VEL
LIN {X 0,Y 460.5,Z 229.618,A -85,B 0,C 180,E1 -8069.755,E2 -8069.755} C_VEL
LIN {X 0,Y 460.486,Z 229.624,A -85,B 0,C 180,E1 -8072.746,E2 -8072.746} C_VEL
LIN {X 0,Y 460.509,Z 229.618,A -85,B 0,C 180,E1 -8075.661,E2 -8075.661} C_VEL
LIN {X 0,Y 460.512,Z 229.621,A -85,B 0,C 180,E1 -8078.575,E2 -8078.575} C_VEL
LIN {X 0,Y 460.523,Z 229.618,A -85,B 0,C 180,E1 -8081.303,E2 -8081.303} C_VEL
LIN {X 0,Y 460.559,Z 229.61,A -85,B 0,C 180,E1 -8084.053,E2 -8084.053} C_VEL
LIN {X 0,Y 460.598,Z 229.604,A -85,B 0,C 180,E1 -8087.661,E2 -8087.661} C_VEL
LIN {X 0,Y 460.591,Z 229.611,A -85,B 0,C 180,E1 -8091.218,E2 -8091.218} C_VEL
LIN {X 0,Y 460.672,Z 229.596,A -85,B 0,C 180,E1 -8093.864,E2 -8093.864} C_VEL
LIN {X 0,Y 460.747,Z 229.592,A -85,B 0,C 180,E1 -8097.372,E2 -8097.372} C_VEL
LIN {X 0,Y 460.83,Z 229.577,A -85,B 0,C 180,E1 -8099.994,E2 -8099.994} C_VEL
LIN {X 0,Y 460.778,Z 229.584,A -85,B 0,C 180,E1 -8102.617,E2 -8102.617} C_VEL
LIN {X 0,Y 460.664,Z 229.6,A -85,B 0,C 180,E1 -8106.124,E2 -8106.124} C_VEL
LIN {X 0,Y 460.604,Z 229.608,A -85,B 0,C 180,E1 -8108.77,E2 -8108.77} C_VEL
LIN {X 0,Y 460.606,Z 229.607,A -85,B 0,C 180,E1 -8112.451,E2 -8112.451} C_VEL
LIN {X 0,Y 460.568,Z 229.617,A -85,B 0,C 180,E1 -8115.992,E2 -8115.992} C_VEL
LIN {X 0,Y 460.537,Z 229.618,A -85,B 0,C 180,E1 -8118.896,E2 -8118.896} C_VEL
LIN {X 0,Y 460.528,Z 229.622,A -85,B 0,C 180,E1 -8121.477,E2 -8121.477} C_VEL
LIN {X 0,Y 460.582,Z 229.734,A -85,B 0,C 180,E1 -8123.431,E2 -8123.431} C_VEL
LIN {X 0,Y 461.843,Z 236.036,A -85,B 0,C 180,E1 -8124.73,E2 -8124.73} C_VEL
LIN {X 0,Y 461.926,Z 241.017,A -85,B 0,C 180,E1 -8125.66,E2 -8125.66} C_VEL
LIN {X 0,Y 461.442,Z 257.463,A -85,B 0,C 180,E1 -8128.677,E2 -8128.677} C_VEL
LIN {X 0,Y 461.925,Z 260.155,A -85,B 0,C 180,E1 -8128.784,E2 -8128.784} C_VEL
LIN {X 0,Y 464.59,Z 275.452,A -85,B 0,C 180,E1 -8129.148,E2 -8129.148} C_VEL
LIN {X 0,Y 463.659,Z 365.944,A -85,B 0,C 180,E1 -8130.635,E2 -8130.635} C_VEL
LIN {X 0,Y 463.304,Z 379.475,A -85,B 0,C 180,E1 -8131.039,E2 -8131.039} C_VEL
LIN {X 0,Y 462.962,Z 391.997,A -85,B 0,C 180,E1 -8131.595,E2 -8131.595} C_VEL
LIN {X 0,Y 462.51,Z 403.004,A -85,B 0,C 180,E1 -8132.249,E2 -8132.249} C_VEL
LIN {X 0,Y 461.962,Z 414.466,A -85,B 0,C 180,E1 -8133.12,E2 -8133.12} C_VEL
LIN {X 0,Y 461.399,Z 425.392,A -85,B 0,C 180,E1 -8134.162,E2 -8134.162} C_VEL
LIN {X 0,Y 460.914,Z 434.142,A -85,B 0,C 180,E1 -8135.194,E2 -8135.194} C_VEL
LIN {X 0,Y 460.454,Z 443.237,A -85,B 0,C 180,E1 -8136.521,E2 -8136.521} C_VEL
LIN {X 0,Y 460.096,Z 450.967,A -85,B 0,C 180,E1 -8137.928,E2 -8137.928} C_VEL
LIN {X 0,Y 459.834,Z 457.097,A -85,B 0,C 180,E1 -8139.355,E2 -8139.355} C_VEL
LIN {X 0,Y 459.688,Z 461.283,A -85,B 0,C 180,E1 -8140.59,E2 -8140.59} C_VEL
LIN {X 0,Y 459.507,Z 465.465,A -85,B 0,C 180,E1 -8142.285,E2 -8142.285} C_VEL
LIN {X 0,Y 459.437,Z 468.111,A -85,B 0,C 180,E1 -8144.034,E2 -8144.034} C_VEL
LIN {X 0,Y 459.424,Z 469.003,A -85,B 0,C 180,E1 -8145.28,E2 -8145.28} C_VEL
LIN {X 0,Y 459.382,Z 469.066,A -85,B 0,C 180,E1 -8146.496,E2 -8146.496} C_VEL
LIN {X 0,Y 459.41,Z 468.39,A -85,B 0,C 180,E1 -8147.695,E2 -8147.695} C_VEL
LIN {X 0,Y 459.477,Z 467.005,A -85,B 0,C 180,E1 -8148.877,E2 -8148.877} C_VEL
LIN {X 0,Y 459.577,Z 463.544,A -85,B 0,C 180,E1 -8150.61,E2 -8150.61} C_VEL
LIN {X 0,Y 459.777,Z 458.457,A -85,B 0,C 180,E1 -8152.31,E2 -8152.31} C_VEL
LIN {X 0,Y 459.996,Z 452.534,A -85,B 0,C 180,E1 -8153.767,E2 -8153.767} C_VEL
LIN {X 0,Y 460.305,Z 445.981,A -85,B 0,C 180,E1 -8155.047,E2 -8155.047} C_VEL
LIN {X 0,Y 460.685,Z 437.173,A -85,B 0,C 180,E1 -8156.428,E2 -8156.428} C_VEL
LIN {X 0,Y 461.215,Z 427.427,A -85,B 0,C 180,E1 -8157.642,E2 -8157.642} C_VEL
LIN {X 0,Y 461.245,Z 426.806,A -85,B 0,C 180,E1 -8157.712,E2 -8157.712} C_VEL
LIN {X 0,Y 460.814,Z 422.409,A -85,B 0,C 180,E1 -8158.2,E2 -8158.2} C_VEL
LIN {X 0,Y 458.387,Z 415.033,A -85,B 0,C 180,E1 -8158.969,E2 -8158.969} C_VEL
LIN {X 0,Y 455.944,Z 407.223,A -85,B 0,C 180,E1 -8159.67,E2 -8159.67} C_VEL
LIN {X 0,Y 455.483,Z 402.146,A -85,B 0,C 180,E1 -8160.045,E2 -8160.045} C_VEL
LIN {X 0,Y 456.021,Z 389.992,A -85,B 0,C 180,E1 -8160.749,E2 -8160.749} C_VEL
LIN {X 0,Y 456.381,Z 377.523,A -85,B 0,C 180,E1 -8161.284,E2 -8161.284} C_VEL
LIN {X 0,Y 456.716,Z 365.323,A -85,B 0,C 180,E1 -8161.636,E2 -8161.636} C_VEL
LIN {X 0,Y 457.47,Z 274.902,A -85,B 0,C 180,E1 -8163.132,E2 -8163.132} C_VEL
LIN {X 0,Y 454.581,Z 258.638,A -85,B 0,C 180,E1 -8163.534,E2 -8163.534} C_VEL
LIN {X 0,Y 454.558,Z 257.366,A -85,B 0,C 180,E1 -8163.712,E2 -8163.712} C_VEL
LIN {X 0,Y 455.358,Z 241.461,A -85,B 0,C 180,E1 -8167.066,E2 -8167.066} C_VEL
LIN {X 0,Y 454.217,Z 234.278,A -85,B 0,C 180,E1 -8168.68,E2 -8168.68} C_VEL
LIN {X 0,Y 453.46,Z 230.553,A -85,B 0,C 180,E1 -8169.593,E2 -8169.593} C_VEL
LIN {X 0,Y 453.435,Z 230.504,A -85,B 0,C 180,E1 -8171.943,E2 -8171.943} C_VEL
LIN {X 0,Y 453.49,Z 230.499,A -85,B 0,C 180,E1 -8174.726,E2 -8174.726} C_VEL
LIN {X 0,Y 453.525,Z 230.487,A -85,B 0,C 180,E1 -8177.472,E2 -8177.472} C_VEL
LIN {X 0,Y 453.522,Z 230.49,A -85,B 0,C 180,E1 -8181.087,E2 -8181.087} C_VEL
LIN {X 0,Y 453.607,Z 230.476,A -85,B 0,C 180,E1 -8183.775,E2 -8183.775} C_VEL
LIN {X 0,Y 453.7,Z 230.468,A -85,B 0,C 180,E1 -8187.338,E2 -8187.338} C_VEL
LIN {X 0,Y 453.745,Z 230.459,A -85,B 0,C 180,E1 -8190.002,E2 -8190.002} C_VEL
LIN {X 0,Y 453.7,Z 230.468,A -85,B 0,C 180,E1 -8192.665,E2 -8192.665} C_VEL
LIN {X 0,Y 453.609,Z 230.476,A -85,B 0,C 180,E1 -8196.228,E2 -8196.228} C_VEL
LIN {X 0,Y 453.525,Z 230.49,A -85,B 0,C 180,E1 -8198.916,E2 -8198.916} C_VEL
LIN {X 0,Y 453.53,Z 230.486,A -85,B 0,C 180,E1 -8202.554,E2 -8202.554} C_VEL
LIN {X 0,Y 453.475,Z 230.494,A -85,B 0,C 180,E1 -8206.2,E2 -8206.2} C_VEL
LIN {X 0,Y 453.45,Z 230.497,A -85,B 0,C 180,E1 -8209.044,E2 -8209.044} C_VEL
LIN {X 0,Y 453.411,Z 230.508,A -85,B 0,C 180,E1 -8211.841,E2 -8211.841} C_VEL
LIN {X 0,Y 453.461,Z 230.495,A -85,B 0,C 180,E1 -8214.739,E2 -8214.739} C_VEL
LIN {X 0,Y 453.477,Z 230.502,A -85,B 0,C 180,E1 -8217.966,E2 -8217.966} C_VEL
LIN {X 0,Y 453.426,Z 230.5,A -85,B 0,C 180,E1 -8220.765,E2 -8220.765} C_VEL
LIN {X 0,Y 453.422,Z 230.505,A -85,B 0,C 180,E1 -8223.919,E2 -8223.919} C_VEL
LIN {X 0,Y 453.418,Z 230.5,A -85,B 0,C 180,E1 -8227.194,E2 -8227.194} C_VEL
LIN {X 0,Y 453.478,Z 230.492,A -85,B 0,C 180,E1 -8229.452,E2 -8229.452} C_VEL
LIN {X 0,Y 453.446,Z 230.498,A -85,B 0,C 180,E1 -8232.998,E2 -8232.998} C_VEL
LIN {X 0,Y 453.434,Z 230.498,A -85,B 0,C 180,E1 -8235.787,E2 -8235.787} C_VEL
LIN {X 0,Y 453.457,Z 230.498,A -85,B 0,C 180,E1 -8238.218,E2 -8238.218} C_VEL
LIN {X 0,Y 453.495,Z 230.498,A -85,B 0,C 180,E1 -8240.795,E2 -8240.795} C_VEL
LIN {X 0,Y 453.423,Z 230.499,A -85,B 0,C 180,E1 -8243.924,E2 -8243.924} C_VEL
LIN {X 0,Y 453.452,Z 230.501,A -85,B 0,C 180,E1 -8247.158,E2 -8247.158} C_VEL
LIN {X 0,Y 453.449,Z 230.496,A -85,B 0,C 180,E1 -8250.275,E2 -8250.275} C_VEL
LIN {X 0,Y 453.482,Z 230.499,A -85,B 0,C 180,E1 -8253.301,E2 -8253.301} C_VEL
LIN {X 0,Y 453.484,Z 230.492,A -85,B 0,C 180,E1 -8256.246,E2 -8256.246} C_VEL
LIN {X 0,Y 453.468,Z 230.499,A -85,B 0,C 180,E1 -8259.125,E2 -8259.125} C_VEL
LIN {X 0,Y 453.491,Z 230.493,A -85,B 0,C 180,E1 -8261.951,E2 -8261.951} C_VEL
LIN {X 0,Y 453.53,Z 230.486,A -85,B 0,C 180,E1 -8264.733,E2 -8264.733} C_VEL
LIN {X 0,Y 453.553,Z 230.484,A -85,B 0,C 180,E1 -8268.386,E2 -8268.386} C_VEL
LIN {X 0,Y 453.582,Z 230.48,A -85,B 0,C 180,E1 -8271.093,E2 -8271.093} C_VEL
LIN {X 0,Y 453.645,Z 230.48,A -85,B 0,C 180,E1 -8273.781,E2 -8273.781} C_VEL
LIN {X 0,Y 453.735,Z 230.462,A -85,B 0,C 180,E1 -8277.343,E2 -8277.343} C_VEL
LIN {X 0,Y 453.772,Z 230.464,A -85,B 0,C 180,E1 -8280.006,E2 -8280.006} C_VEL
LIN {X 0,Y 453.71,Z 230.466,A -85,B 0,C 180,E1 -8282.669,E2 -8282.669} C_VEL
LIN {X 0,Y 453.647,Z 230.48,A -85,B 0,C 180,E1 -8286.231,E2 -8286.231} C_VEL
LIN {X 0,Y 453.572,Z 230.482,A -85,B 0,C 180,E1 -8288.919,E2 -8288.919} C_VEL
LIN {X 0,Y 453.579,Z 230.488,A -85,B 0,C 180,E1 -8292.534,E2 -8292.534} C_VEL
LIN {X 0,Y 453.561,Z 230.485,A -85,B 0,C 180,E1 -8296.2,E2 -8296.2} C_VEL
LIN {X 0,Y 453.534,Z 230.489,A -85,B 0,C 180,E1 -8299.043,E2 -8299.043} C_VEL
LIN {X 0,Y 453.493,Z 230.49,A -85,B 0,C 180,E1 -8301.84,E2 -8301.84} C_VEL
LIN {X 0,Y 453.504,Z 230.496,A -85,B 0,C 180,E1 -8304.74,E2 -8304.74} C_VEL
LIN {X 0,Y 453.481,Z 230.492,A -85,B 0,C 180,E1 -8307.946,E2 -8307.946} C_VEL
LIN {X 0,Y 453.476,Z 230.497,A -85,B 0,C 180,E1 -8310.764,E2 -8310.764} C_VEL
LIN {X 0,Y 453.486,Z 230.492,A -85,B 0,C 180,E1 -8313.916,E2 -8313.916} C_VEL
LIN {X 0,Y 453.469,Z 230.5,A -85,B 0,C 180,E1 -8317.192,E2 -8317.192} C_VEL
LIN {X 0,Y 453.491,Z 230.491,A -85,B 0,C 180,E1 -8320.614,E2 -8320.614} C_VEL
LIN {X 0,Y 453.46,Z 230.496,A -85,B 0,C 180,E1 -8324.226,E2 -8324.226} C_VEL
LIN {X 0,Y 453.435,Z 230.499,A -85,B 0,C 180,E1 -8327,E2 -8327} C_VEL
LIN {X 0,Y 453.491,Z 230.495,A -85,B 0,C 180,E1 -8329.414,E2 -8329.414} C_VEL
LIN {X 0,Y 453.458,Z 230.495,A -85,B 0,C 180,E1 -8332.81,E2 -8332.81} C_VEL
LIN {X 0,Y 453.485,Z 230.499,A -85,B 0,C 180,E1 -8336.087,E2 -8336.087} C_VEL
LIN {X 0,Y 453.478,Z 230.493,A -85,B 0,C 180,E1 -8339.239,E2 -8339.239} C_VEL
LIN {X 0,Y 453.526,Z 230.495,A -85,B 0,C 180,E1 -8342.296,E2 -8342.296} C_VEL
LIN {X 0,Y 453.561,Z 230.622,A -85,B 0,C 180,E1 -8344.655,E2 -8344.655} C_VEL
LIN {X 0,Y 455.657,Z 241.979,A -85,B 0,C 180,E1 -8347.078,E2 -8347.078} C_VEL
LIN {X 0,Y 455.459,Z 249.214,A -85,B 0,C 180,E1 -8348.5,E2 -8348.5} C_VEL
LIN {X 0,Y 454.618,Z 266.071,A -85,B 0,C 180,E1 -8351.756,E2 -8351.756} C_VEL
LIN {X 0,Y 454.454,Z 269.925,A -85,B 0,C 180,E1 -8352.464,E2 -8352.464} C_VEL
LIN {X 0,Y 455.285,Z 275.158,A -85,B 0,C 180,E1 -8352.628,E2 -8352.628} C_VEL
LIN {X 0,Y 457.586,Z 290.154,A -85,B 0,C 180,E1 -8352.962,E2 -8352.962} C_VEL
LIN {X 0,Y 456.704,Z 377.605,A -85,B 0,C 180,E1 -8354.405,E2 -8354.405} C_VEL
LIN {X 0,Y 456.352,Z 390.811,A -85,B 0,C 180,E1 -8354.793,E2 -8354.793} C_VEL
LIN {X 0,Y 455.919,Z 402.972,A -85,B 0,C 180,E1 -8355.321,E2 -8355.321} C_VEL
LIN {X 0,Y 455.339,Z 415.27,A -85,B 0,C 180,E1 -8356.043,E2 -8356.043} C_VEL
LIN {X 0,Y 454.775,Z 426.705,A -85,B 0,C 180,E1 -8356.92,E2 -8356.92} C_VEL
LIN {X 0,Y 454.271,Z 437.358,A -85,B 0,C 180,E1 -8357.943,E2 -8357.943} C_VEL
LIN {X 0,Y 453.715,Z 446.768,A -85,B 0,C 180,E1 -8359.06,E2 -8359.06} C_VEL
LIN {X 0,Y 453.256,Z 455.855,A -85,B 0,C 180,E1 -8360.403,E2 -8360.403} C_VEL
LIN {X 0,Y 452.952,Z 463.176,A -85,B 0,C 180,E1 -8361.747,E2 -8361.747} C_VEL
LIN {X 0,Y 452.732,Z 468.121,A -85,B 0,C 180,E1 -8362.865,E2 -8362.865} C_VEL
LIN {X 0,Y 452.596,Z 472.921,A -85,B 0,C 180,E1 -8364.206,E2 -8364.206} C_VEL
LIN {X 0,Y 452.493,Z 476.59,A -85,B 0,C 180,E1 -8365.545,E2 -8365.545} C_VEL
LIN {X 0,Y 452.46,Z 478.485,A -85,B 0,C 180,E1 -8366.436,E2 -8366.436} C_VEL
LIN {X 0,Y 452.496,Z 479.914,A -85,B 0,C 180,E1 -8367.328,E2 -8367.328} C_VEL
LIN {X 0,Y 452.408,Z 481.546,A -85,B 0,C 180,E1 -8369.108,E2 -8369.108} C_VEL
LIN {X 0,Y 452.412,Z 481.775,A -85,B 0,C 180,E1 -8369.998,E2 -8369.998} C_VEL
LIN {X 0,Y 452.408,Z 481.567,A -85,B 0,C 180,E1 -8370.889,E2 -8370.889} C_VEL
LIN {X 0,Y 452.495,Z 479.961,A -85,B 0,C 180,E1 -8372.669,E2 -8372.669} C_VEL
LIN {X 0,Y 452.459,Z 478.558,A -85,B 0,C 180,E1 -8373.561,E2 -8373.561} C_VEL
LIN {X 0,Y 452.559,Z 475.607,A -85,B 0,C 180,E1 -8374.898,E2 -8374.898} C_VEL
LIN {X 0,Y 452.622,Z 471.066,A -85,B 0,C 180,E1 -8376.394,E2 -8376.394} C_VEL
LIN {X 0,Y 452.867,Z 465.455,A -85,B 0,C 180,E1 -8377.803,E2 -8377.803} C_VEL
LIN {X 0,Y 453.15,Z 458.729,A -85,B 0,C 180,E1 -8379.145,E2 -8379.145} C_VEL
LIN {X 0,Y 453.578,Z 450.384,A -85,B 0,C 180,E1 -8380.488,E2 -8380.488} C_VEL
LIN {X 0,Y 454.08,Z 441.812,A -85,B 0,C 180,E1 -8381.606,E2 -8381.606} C_VEL
LIN {X 0,Y 454.633,Z 431.982,A -85,B 0,C 180,E1 -8382.653,E2 -8382.653} C_VEL
LIN {X 0,Y 455.138,Z 420.78,A -85,B 0,C 180,E1 -8383.618,E2 -8383.618} C_VEL
LIN {X 0,Y 455.702,Z 409.285,A -85,B 0,C 180,E1 -8384.398,E2 -8384.398} C_VEL
LIN {X 0,Y 456.215,Z 397.401,A -85,B 0,C 180,E1 -8385.009,E2 -8385.009} C_VEL
LIN {X 0,Y 456.676,Z 383.743,A -85,B 0,C 180,E1 -8385.507,E2 -8385.507} C_VEL
LIN {X 0,Y 456.95,Z 371.514,A -85,B 0,C 180,E1 -8385.784,E2 -8385.784} C_VEL
LIN {X 0,Y 457.705,Z 288.665,A -85,B 0,C 180,E1 -8387.15,E2 -8387.15} C_VEL
LIN {X 0,Y 454.529,Z 269.659,A -85,B 0,C 180,E1 -8387.628,E2 -8387.628} C_VEL
LIN {X 0,Y 455.126,Z 253.839,A -85,B 0,C 180,E1 -8390.565,E2 -8390.565} C_VEL
LIN {X 0,Y 455.684,Z 242.71,A -85,B 0,C 180,E1 -8392.677,E2 -8392.677} C_VEL
LIN {X 0,Y 453.982,Z 232.791,A -85,B 0,C 180,E1 -8394.705,E2 -8394.705} C_VEL
LIN {X 0,Y 453.514,Z 230.58,A -85,B 0,C 180,E1 -8395.222,E2 -8395.222} C_VEL
LIN {X 0,Y 453.537,Z 230.493,A -85,B 0,C 180,E1 -8397.956,E2 -8397.956} C_VEL
LIN {X 0,Y 453.473,Z 230.499,A -85,B 0,C 180,E1 -8401.522,E2 -8401.522} C_VEL
LIN {X 0,Y 453.493,Z 230.494,A -85,B 0,C 180,E1 -8404.774,E2 -8404.774} C_VEL
LIN {X 0,Y 453.461,Z 230.501,A -85,B 0,C 180,E1 -8408.309,E2 -8408.309} C_VEL
LIN {X 0,Y 453.475,Z 230.496,A -85,B 0,C 180,E1 -8410.608,E2 -8410.608} C_VEL
LIN {X 0,Y 453.462,Z 230.503,A -85,B 0,C 180,E1 -8414.219,E2 -8414.219} C_VEL
LIN {X 0,Y 453.424,Z 230.501,A -85,B 0,C 180,E1 -8416.996,E2 -8416.996} C_VEL
LIN {X 0,Y 453.473,Z 230.495,A -85,B 0,C 180,E1 -8419.409,E2 -8419.409} C_VEL
LIN {X 0,Y 453.436,Z 230.5,A -85,B 0,C 180,E1 -8422.804,E2 -8422.804} C_VEL
LIN {X 0,Y 453.465,Z 230.5,A -85,B 0,C 180,E1 -8426.082,E2 -8426.082} C_VEL
LIN {X 0,Y 453.456,Z 230.496,A -85,B 0,C 180,E1 -8429.235,E2 -8429.235} C_VEL
LIN {X 0,Y 453.47,Z 230.499,A -85,B 0,C 180,E1 -8432.289,E2 -8432.289} C_VEL
LIN {X 0,Y 453.463,Z 230.497,A -85,B 0,C 180,E1 -8435.258,E2 -8435.258} C_VEL
LIN {X 0,Y 453.472,Z 230.496,A -85,B 0,C 180,E1 -8438.412,E2 -8438.412} C_VEL
LIN {X 0,Y 453.479,Z 230.496,A -85,B 0,C 180,E1 -8441.002,E2 -8441.002} C_VEL
LIN {X 0,Y 453.505,Z 230.492,A -85,B 0,C 180,E1 -8444.72,E2 -8444.72} C_VEL
LIN {X 0,Y 453.544,Z 230.483,A -85,B 0,C 180,E1 -8448.373,E2 -8448.373} C_VEL
LIN {X 0,Y 453.558,Z 230.487,A -85,B 0,C 180,E1 -8451.081,E2 -8451.081} C_VEL
LIN {X 0,Y 453.639,Z 230.472,A -85,B 0,C 180,E1 -8453.769,E2 -8453.769} C_VEL
LIN {X 0,Y 453.694,Z 230.471,A -85,B 0,C 180,E1 -8457.331,E2 -8457.331} C_VEL
LIN {X 0,Y 453.8,Z 230.453,A -85,B 0,C 180,E1 -8459.994,E2 -8459.994} C_VEL
LIN {X 0,Y 453.722,Z 230.463,A -85,B 0,C 180,E1 -8462.657,E2 -8462.657} C_VEL
LIN {X 0,Y 453.63,Z 230.476,A -85,B 0,C 180,E1 -8466.22,E2 -8466.22} C_VEL
LIN {X 0,Y 453.567,Z 230.485,A -85,B 0,C 180,E1 -8468.907,E2 -8468.907} C_VEL
LIN {X 0,Y 453.574,Z 230.483,A -85,B 0,C 180,E1 -8472.545,E2 -8472.545} C_VEL
LIN {X 0,Y 453.513,Z 230.494,A -85,B 0,C 180,E1 -8476.19,E2 -8476.19} C_VEL
LIN {X 0,Y 453.486,Z 230.497,A -85,B 0,C 180,E1 -8479.035,E2 -8479.035} C_VEL
LIN {X 0,Y 453.469,Z 230.501,A -85,B 0,C 180,E1 -8481.829,E2 -8481.829} C_VEL
LIN {X 0,Y 453.511,Z 230.608,A -85,B 0,C 180,E1 -8483.208,E2 -8483.208} C_VEL
LIN {X 0,Y 455.101,Z 238.692,A -85,B 0,C 180,E1 -8484.878,E2 -8484.878} C_VEL
LIN {X 0,Y 454.532,Z 256.486,A -85,B 0,C 180,E1 -8488.201,E2 -8488.201} C_VEL
LIN {X 0,Y 454.569,Z 257.986,A -85,B 0,C 180,E1 -8488.426,E2 -8488.426} C_VEL
LIN {X 0,Y 457.844,Z 275.774,A -85,B 0,C 180,E1 -8488.882,E2 -8488.882} C_VEL
LIN {X 0,Y 456.84,Z 366.125,A -85,B 0,C 180,E1 -8490.392,E2 -8490.392} C_VEL
LIN {X 0,Y 456.481,Z 379.936,A -85,B 0,C 180,E1 -8490.815,E2 -8490.815} C_VEL
LIN {X 0,Y 456.087,Z 392.589,A -85,B 0,C 180,E1 -8491.392,E2 -8491.392} C_VEL
LIN {X 0,Y 455.597,Z 403.646,A -85,B 0,C 180,E1 -8492.067,E2 -8492.067} C_VEL
LIN {X 0,Y 455.005,Z 415.088,A -85,B 0,C 180,E1 -8492.959,E2 -8492.959} C_VEL
LIN {X 0,Y 454.449,Z 425.314,A -85,B 0,C 180,E1 -8493.954,E2 -8493.954} C_VEL
LIN {X 0,Y 453.895,Z 434.657,A -85,B 0,C 180,E1 -8495.078,E2 -8495.078} C_VEL
LIN {X 0,Y 453.397,Z 443.987,A -85,B 0,C 180,E1 -8496.476,E2 -8496.476} C_VEL
LIN {X 0,Y 453.094,Z 450.67,A -85,B 0,C 180,E1 -8497.718,E2 -8497.718} C_VEL
LIN {X 0,Y 452.787,Z 456.667,A -85,B 0,C 180,E1 -8499.1,E2 -8499.1} C_VEL
LIN {X 0,Y 452.6,Z 461.927,A -85,B 0,C 180,E1 -8500.695,E2 -8500.695} C_VEL
LIN {X 0,Y 452.446,Z 464.916,A -85,B 0,C 180,E1 -8501.896,E2 -8501.896} C_VEL
LIN {X 0,Y 452.378,Z 467.114,A -85,B 0,C 180,E1 -8503.111,E2 -8503.111} C_VEL
LIN {X 0,Y 452.33,Z 468.558,A -85,B 0,C 180,E1 -8504.383,E2 -8504.383} C_VEL
LIN {X 0,Y 452.322,Z 469.186,A -85,B 0,C 180,E1 -8505.641,E2 -8505.641} C_VEL
LIN {X 0,Y 452.304,Z 469.029,A -85,B 0,C 180,E1 -8506.898,E2 -8506.898} C_VEL
LIN {X 0,Y 452.333,Z 468.01,A -85,B 0,C 180,E1 -8508.213,E2 -8508.213} C_VEL
LIN {X 0,Y 452.404,Z 466.038,A -85,B 0,C 180,E1 -8509.557,E2 -8509.557} C_VEL
LIN {X 0,Y 452.53,Z 463.014,A -85,B 0,C 180,E1 -8510.929,E2 -8510.929} C_VEL
LIN {X 0,Y 452.7,Z 458.773,A -85,B 0,C 180,E1 -8512.335,E2 -8512.335} C_VEL
LIN {X 0,Y 452.946,Z 452.64,A -85,B 0,C 180,E1 -8513.873,E2 -8513.873} C_VEL
LIN {X 0,Y 453.307,Z 445.71,A -85,B 0,C 180,E1 -8515.24,E2 -8515.24} C_VEL
LIN {X 0,Y 453.621,Z 438.165,A -85,B 0,C 180,E1 -8516.448,E2 -8516.448} C_VEL
LIN {X 0,Y 454.139,Z 429.33,A -85,B 0,C 180,E1 -8517.602,E2 -8517.602} C_VEL
LIN {X 0,Y 454.649,Z 419.103,A -85,B 0,C 180,E1 -8518.685,E2 -8518.685} C_VEL
LIN {X 0,Y 455.22,Z 408.183,A -85,B 0,C 180,E1 -8519.615,E2 -8519.615} C_VEL
LIN {X 0,Y 455.483,Z 402.146,A -85,B 0,C 180,E1 -8520.045,E2 -8520.045} C_VEL
LIN {X 0,Y 455.064,Z 396.944,A -85,B 0,C 180,E1 -8520.394,E2 -8520.394} C_VEL
LIN {X 0,Y 452.729,Z 388.36,A -85,B 0,C 180,E1 -8520.943,E2 -8520.943} C_VEL
LIN {X 0,Y 450.273,Z 379.51,A -85,B 0,C 180,E1 -8521.411,E2 -8521.411} C_VEL
LIN {X 0,Y 449.645,Z 373.893,A -85,B 0,C 180,E1 -8521.63,E2 -8521.63} C_VEL
LIN {X 0,Y 449.925,Z 360.343,A -85,B 0,C 180,E1 -8521.963,E2 -8521.963} C_VEL
LIN {X 0,Y 450.653,Z 275.764,A -85,B 0,C 180,E1 -8523.371,E2 -8523.371} C_VEL
LIN {X 0,Y 447.618,Z 258.59,A -85,B 0,C 180,E1 -8523.804,E2 -8523.804} C_VEL
LIN {X 0,Y 447.779,Z 253.012,A -85,B 0,C 180,E1 -8524.929,E2 -8524.929} C_VEL
LIN {X 0,Y 448.403,Z 242.533,A -85,B 0,C 180,E1 -8527.177,E2 -8527.177} C_VEL
LIN {X 0,Y 446.799,Z 233.402,A -85,B 0,C 180,E1 -8529.275,E2 -8529.275} C_VEL
LIN {X 0,Y 446.42,Z 231.401,A -85,B 0,C 180,E1 -8529.828,E2 -8529.828} C_VEL
LIN {X 0,Y 446.42,Z 231.373,A -85,B 0,C 180,E1 -8533.54,E2 -8533.54} C_VEL
LIN {X 0,Y 446.433,Z 231.376,A -85,B 0,C 180,E1 -8536.343,E2 -8536.343} C_VEL
LIN {X 0,Y 446.43,Z 231.373,A -85,B 0,C 180,E1 -8539.112,E2 -8539.112} C_VEL
LIN {X 0,Y 446.581,Z 231.356,A -85,B 0,C 180,E1 -8542.428,E2 -8542.428} C_VEL
LIN {X 0,Y 446.578,Z 231.357,A -85,B 0,C 180,E1 -8544.583,E2 -8544.583} C_VEL
LIN {X 0,Y 446.644,Z 231.347,A -85,B 0,C 180,E1 -8547.296,E2 -8547.296} C_VEL
LIN {X 0,Y 446.716,Z 231.335,A -85,B 0,C 180,E1 -8550.002,E2 -8550.002} C_VEL
LIN {X 0,Y 446.644,Z 231.347,A -85,B 0,C 180,E1 -8552.707,E2 -8552.707} C_VEL
LIN {X 0,Y 446.577,Z 231.352,A -85,B 0,C 180,E1 -8556.326,E2 -8556.326} C_VEL
LIN {X 0,Y 446.471,Z 231.37,A -85,B 0,C 180,E1 -8559.058,E2 -8559.058} C_VEL
LIN {X 0,Y 446.464,Z 231.367,A -85,B 0,C 180,E1 -8562.733,E2 -8562.733} C_VEL
LIN {X 0,Y 446.426,Z 231.372,A -85,B 0,C 180,E1 -8566.232,E2 -8566.232} C_VEL
LIN {X 0,Y 446.401,Z 231.378,A -85,B 0,C 180,E1 -8569.308,E2 -8569.308} C_VEL
LIN {X 0,Y 446.352,Z 231.383,A -85,B 0,C 180,E1 -8572.204,E2 -8572.204} C_VEL
LIN {X 0,Y 446.408,Z 231.374,A -85,B 0,C 180,E1 -8575.157,E2 -8575.157} C_VEL
LIN {X 0,Y 446.425,Z 231.377,A -85,B 0,C 180,E1 -8578.184,E2 -8578.184} C_VEL
LIN {X 0,Y 446.374,Z 231.378,A -85,B 0,C 180,E1 -8581.305,E2 -8581.305} C_VEL
LIN {X 0,Y 446.376,Z 231.381,A -85,B 0,C 180,E1 -8584.529,E2 -8584.529} C_VEL
LIN {X 0,Y 446.384,Z 231.382,A -85,B 0,C 180,E1 -8588.089,E2 -8588.089} C_VEL
LIN {X 0,Y 446.4,Z 231.376,A -85,B 0,C 180,E1 -8590.927,E2 -8590.927} C_VEL
LIN {X 0,Y 446.4,Z 231.375,A -85,B 0,C 180,E1 -8593.847,E2 -8593.847} C_VEL
LIN {X 0,Y 446.405,Z 231.38,A -85,B 0,C 180,E1 -8596.404,E2 -8596.404} C_VEL
LIN {X 0,Y 446.432,Z 231.37,A -85,B 0,C 180,E1 -8599.812,E2 -8599.812} C_VEL
LIN {X 0,Y 446.398,Z 231.375,A -85,B 0,C 180,E1 -8602.131,E2 -8602.131} C_VEL
LIN {X 0,Y 446.398,Z 231.376,A -85,B 0,C 180,E1 -8605.484,E2 -8605.484} C_VEL
LIN {X 0,Y 446.388,Z 231.38,A -85,B 0,C 180,E1 -8608.707,E2 -8608.707} C_VEL
LIN {X 0,Y 446.462,Z 231.367,A -85,B 0,C 180,E1 -8611.829,E2 -8611.829} C_VEL
LIN {X 0,Y 446.429,Z 231.374,A -85,B 0,C 180,E1 -8614.854,E2 -8614.854} C_VEL
LIN {X 0,Y 446.433,Z 231.37,A -85,B 0,C 180,E1 -8618.252,E2 -8618.252} C_VEL
LIN {X 0,Y 446.44,Z 231.375,A -85,B 0,C 180,E1 -8621.656,E2 -8621.656} C_VEL
LIN {X 0,Y 446.499,Z 231.362,A -85,B 0,C 180,E1 -8624.487,E2 -8624.487} C_VEL
LIN {X 0,Y 446.511,Z 231.362,A -85,B 0,C 180,E1 -8628.2,E2 -8628.2} C_VEL
LIN {X 0,Y 446.53,Z 231.358,A -85,B 0,C 180,E1 -8630.951,E2 -8630.951} C_VEL
LIN {X 0,Y 446.614,Z 231.354,A -85,B 0,C 180,E1 -8633.682,E2 -8633.682} C_VEL
LIN {X 0,Y 446.682,Z 231.34,A -85,B 0,C 180,E1 -8637.301,E2 -8637.301} C_VEL
LIN {X 0,Y 446.723,Z 231.342,A -85,B 0,C 180,E1 -8640.006,E2 -8640.006} C_VEL
LIN {X 0,Y 446.66,Z 231.344,A -85,B 0,C 180,E1 -8642.711,E2 -8642.711} C_VEL
LIN {X 0,Y 446.616,Z 231.355,A -85,B 0,C 180,E1 -8646.33,E2 -8646.33} C_VEL
LIN {X 0,Y 446.524,Z 231.36,A -85,B 0,C 180,E1 -8649.061,E2 -8649.061} C_VEL
LIN {X 0,Y 446.536,Z 231.362,A -85,B 0,C 180,E1 -8652.734,E2 -8652.734} C_VEL
LIN {X 0,Y 446.505,Z 231.368,A -85,B 0,C 180,E1 -8656.463,E2 -8656.463} C_VEL
LIN {X 0,Y 446.485,Z 231.365,A -85,B 0,C 180,E1 -8659.307,E2 -8659.307} C_VEL
LIN {X 0,Y 446.434,Z 231.371,A -85,B 0,C 180,E1 -8662.204,E2 -8662.204} C_VEL
LIN {X 0,Y 446.447,Z 231.373,A -85,B 0,C 180,E1 -8665.158,E2 -8665.158} C_VEL
LIN {X 0,Y 446.436,Z 231.37,A -85,B 0,C 180,E1 -8668.187,E2 -8668.187} C_VEL
LIN {X 0,Y 446.428,Z 231.377,A -85,B 0,C 180,E1 -8671.304,E2 -8671.304} C_VEL
LIN {X 0,Y 446.441,Z 231.37,A -85,B 0,C 180,E1 -8674.526,E2 -8674.526} C_VEL
LIN {X 0,Y 446.43,Z 231.371,A -85,B 0,C 180,E1 -8678.08,E2 -8678.08} C_VEL
LIN {X 0,Y 446.42,Z 231.379,A -85,B 0,C 180,E1 -8681.396,E2 -8681.396} C_VEL
LIN {X 0,Y 446.435,Z 231.372,A -85,B 0,C 180,E1 -8685.11,E2 -8685.11} C_VEL
LIN {X 0,Y 446.42,Z 231.372,A -85,B 0,C 180,E1 -8688.607,E2 -8688.607} C_VEL
LIN {X 0,Y 446.419,Z 231.379,A -85,B 0,C 180,E1 -8691.925,E2 -8691.925} C_VEL
LIN {X 0,Y 446.441,Z 231.372,A -85,B 0,C 180,E1 -8695.477,E2 -8695.477} C_VEL
LIN {X 0,Y 446.429,Z 231.373,A -85,B 0,C 180,E1 -8698.699,E2 -8698.699} C_VEL
LIN {X 0,Y 446.469,Z 231.373,A -85,B 0,C 180,E1 -8701.83,E2 -8701.83} C_VEL
LIN {X 0,Y 446.519,Z 231.58,A -85,B 0,C 180,E1 -8704.476,E2 -8704.476} C_VEL
LIN {X 0,Y 448.674,Z 243.03,A -85,B 0,C 180,E1 -8706.945,E2 -8706.945} C_VEL
LIN {X 0,Y 448.554,Z 249.063,A -85,B 0,C 180,E1 -8708.152,E2 -8708.152} C_VEL
LIN {X 0,Y 447.677,Z 265.9,A -85,B 0,C 180,E1 -8711.463,E2 -8711.463} C_VEL
LIN {X 0,Y 447.503,Z 270.022,A -85,B 0,C 180,E1 -8712.213,E2 -8712.213} C_VEL
LIN {X 0,Y 449.027,Z 279.237,A -85,B 0,C 180,E1 -8712.466,E2 -8712.466} C_VEL
LIN {X 0,Y 450.742,Z 291.395,A -85,B 0,C 180,E1 -8712.737,E2 -8712.737} C_VEL
LIN {X 0,Y 449.843,Z 378.005,A -85,B 0,C 180,E1 -8714.19,E2 -8714.19} C_VEL
LIN {X 0,Y 449.427,Z 391.8,A -85,B 0,C 180,E1 -8714.611,E2 -8714.611} C_VEL
LIN {X 0,Y 448.895,Z 404.751,A -85,B 0,C 180,E1 -8715.202,E2 -8715.202} C_VEL
LIN {X 0,Y 448.336,Z 416.545,A -85,B 0,C 180,E1 -8715.937,E2 -8715.937} C_VEL
LIN {X 0,Y 447.794,Z 428.23,A -85,B 0,C 180,E1 -8716.872,E2 -8716.872} C_VEL
LIN {X 0,Y 447.246,Z 438.177,A -85,B 0,C 180,E1 -8717.866,E2 -8717.866} C_VEL
LIN {X 0,Y 446.603,Z 448.206,A -85,B 0,C 180,E1 -8719.114,E2 -8719.114} C_VEL
LIN {X 0,Y 446.159,Z 457.039,A -85,B 0,C 180,E1 -8720.478,E2 -8720.478} C_VEL
LIN {X 0,Y 445.859,Z 464.083,A -85,B 0,C 180,E1 -8721.843,E2 -8721.843} C_VEL
LIN {X 0,Y 445.595,Z 469.715,A -85,B 0,C 180,E1 -8723.206,E2 -8723.206} C_VEL
LIN {X 0,Y 445.514,Z 474.134,A -85,B 0,C 180,E1 -8724.567,E2 -8724.567} C_VEL
LIN {X 0,Y 445.42,Z 476.466,A -85,B 0,C 180,E1 -8725.474,E2 -8725.474} C_VEL
LIN {X 0,Y 445.359,Z 478.366,A -85,B 0,C 180,E1 -8726.379,E2 -8726.379} C_VEL
LIN {X 0,Y 445.404,Z 479.803,A -85,B 0,C 180,E1 -8727.285,E2 -8727.285} C_VEL
LIN {X 0,Y 445.357,Z 480.819,A -85,B 0,C 180,E1 -8728.19,E2 -8728.19} C_VEL
LIN {X 0,Y 445.321,Z 481.675,A -85,B 0,C 180,E1 -8729.998,E2 -8729.998} C_VEL
LIN {X 0,Y 445.32,Z 481.473,A -85,B 0,C 180,E1 -8730.903,E2 -8730.903} C_VEL
LIN {X 0,Y 445.357,Z 480.867,A -85,B 0,C 180,E1 -8731.807,E2 -8731.807} C_VEL
LIN {X 0,Y 445.403,Z 479.87,A -85,B 0,C 180,E1 -8732.712,E2 -8732.712} C_VEL
LIN {X 0,Y 445.359,Z 478.469,A -85,B 0,C 180,E1 -8733.617,E2 -8733.617} C_VEL
LIN {X 0,Y 445.491,Z 475.519,A -85,B 0,C 180,E1 -8734.976,E2 -8734.976} C_VEL
LIN {X 0,Y 445.586,Z 470.084,A -85,B 0,C 180,E1 -8736.746,E2 -8736.746} C_VEL
LIN {X 0,Y 445.853,Z 464.362,A -85,B 0,C 180,E1 -8738.154,E2 -8738.154} C_VEL
LIN {X 0,Y 446.198,Z 457.421,A -85,B 0,C 180,E1 -8739.518,E2 -8739.518} C_VEL
LIN {X 0,Y 446.631,Z 448.73,A -85,B 0,C 180,E1 -8740.883,E2 -8740.883} C_VEL
LIN {X 0,Y 447.244,Z 439.823,A -85,B 0,C 180,E1 -8742.016,E2 -8742.016} C_VEL
LIN {X 0,Y 447.857,Z 429.644,A -85,B 0,C 180,E1 -8743.074,E2 -8743.074} C_VEL
LIN {X 0,Y 448.307,Z 419.338,A -85,B 0,C 180,E1 -8743.946,E2 -8743.946} C_VEL
LIN {X 0,Y 448.925,Z 407.347,A -85,B 0,C 180,E1 -8744.736,E2 -8744.736} C_VEL
LIN {X 0,Y 449.52,Z 394.897,A -85,B 0,C 180,E1 -8745.354,E2 -8745.354} C_VEL
LIN {X 0,Y 449.902,Z 382.013,A -85,B 0,C 180,E1 -8745.805,E2 -8745.805} C_VEL
LIN {X 0,Y 450.26,Z 366.775,A -85,B 0,C 180,E1 -8746.112,E2 -8746.112} C_VEL
LIN {X 0,Y 450.911,Z 289.384,A -85,B 0,C 180,E1 -8747.417,E2 -8747.417} C_VEL
LIN {X 0,Y 447.581,Z 269.439,A -85,B 0,C 180,E1 -8747.939,E2 -8747.939} C_VEL
LIN {X 0,Y 448.258,Z 253.812,A -85,B 0,C 180,E1 -8750.895,E2 -8750.895} C_VEL
LIN {X 0,Y 448.769,Z 244.552,A -85,B 0,C 180,E1 -8752.678,E2 -8752.678} C_VEL
LIN {X 0,Y 447.504,Z 236.374,A -85,B 0,C 180,E1 -8754.367,E2 -8754.367} C_VEL
LIN {X 0,Y 446.472,Z 231.408,A -85,B 0,C 180,E1 -8755.492,E2 -8755.492} C_VEL
LIN {X 0,Y 446.495,Z 231.37,A -85,B 0,C 180,E1 -8758.176,E2 -8758.176} C_VEL
LIN {X 0,Y 446.426,Z 231.38,A -85,B 0,C 180,E1 -8761.771,E2 -8761.771} C_VEL
LIN {X 0,Y 446.434,Z 231.374,A -85,B 0,C 180,E1 -8764.52,E2 -8764.52} C_VEL
LIN {X 0,Y 446.415,Z 231.381,A -85,B 0,C 180,E1 -8768.075,E2 -8768.075} C_VEL
LIN {X 0,Y 446.406,Z 231.375,A -85,B 0,C 180,E1 -8771.391,E2 -8771.391} C_VEL
LIN {X 0,Y 446.425,Z 231.372,A -85,B 0,C 180,E1 -8775.104,E2 -8775.104} C_VEL
LIN {X 0,Y 446.402,Z 231.38,A -85,B 0,C 180,E1 -8778.602,E2 -8778.602} C_VEL
LIN {X 0,Y 446.398,Z 231.378,A -85,B 0,C 180,E1 -8781.92,E2 -8781.92} C_VEL
LIN {X 0,Y 446.42,Z 231.374,A -85,B 0,C 180,E1 -8785.472,E2 -8785.472} C_VEL
LIN {X 0,Y 446.408,Z 231.379,A -85,B 0,C 180,E1 -8788.695,E2 -8788.695} C_VEL
LIN {X 0,Y 446.422,Z 231.374,A -85,B 0,C 180,E1 -8791.832,E2 -8791.832} C_VEL
LIN {X 0,Y 446.415,Z 231.38,A -85,B 0,C 180,E1 -8794.841,E2 -8794.841} C_VEL
LIN {X 0,Y 446.441,Z 231.37,A -85,B 0,C 180,E1 -8798.242,E2 -8798.242} C_VEL
LIN {X 0,Y 446.405,Z 231.374,A -85,B 0,C 180,E1 -8801.642,E2 -8801.642} C_VEL
LIN {X 0,Y 446.446,Z 231.371,A -85,B 0,C 180,E1 -8804.473,E2 -8804.473} C_VEL
LIN {X 0,Y 446.507,Z 231.361,A -85,B 0,C 180,E1 -8807.379,E2 -8807.379} C_VEL
LIN {X 0,Y 446.506,Z 231.366,A -85,B 0,C 180,E1 -8810.939,E2 -8810.939} C_VEL
LIN {X 0,Y 446.608,Z 231.349,A -85,B 0,C 180,E1 -8813.67,E2 -8813.67} C_VEL
LIN {X 0,Y 446.643,Z 231.349,A -85,B 0,C 180,E1 -8817.289,E2 -8817.289} C_VEL
LIN {X 0,Y 446.77,Z 231.329,A -85,B 0,C 180,E1 -8819.994,E2 -8819.994} C_VEL
LIN {X 0,Y 446.67,Z 231.342,A -85,B 0,C 180,E1 -8822.699,E2 -8822.699} C_VEL
LIN {X 0,Y 446.598,Z 231.352,A -85,B 0,C 180,E1 -8826.318,E2 -8826.318} C_VEL
LIN {X 0,Y 446.513,Z 231.366,A -85,B 0,C 180,E1 -8829.049,E2 -8829.049} C_VEL
LIN {X 0,Y 446.507,Z 231.364,A -85,B 0,C 180,E1 -8832.723,E2 -8832.723} C_VEL
LIN {X 0,Y 446.458,Z 231.371,A -85,B 0,C 180,E1 -8836.453,E2 -8836.453} C_VEL
LIN {X 0,Y 446.436,Z 231.375,A -85,B 0,C 180,E1 -8839.297,E2 -8839.297} C_VEL
LIN {X 0,Y 446.414,Z 231.38,A -85,B 0,C 180,E1 -8842.192,E2 -8842.192} C_VEL
LIN {X 0,Y 446.465,Z 231.528,A -85,B 0,C 180,E1 -8842.983,E2 -8842.983} C_VEL
LIN {X 0,Y 448.204,Z 240.412,A -85,B 0,C 180,E1 -8844.84,E2 -8844.84} C_VEL
LIN {X 0,Y 447.592,Z 257.714,A -85,B 0,C 180,E1 -8848.094,E2 -8848.094} C_VEL
LIN {X 0,Y 448.671,Z 263.209,A -85,B 0,C 180,E1 -8848.271,E2 -8848.271} C_VEL
LIN {X 0,Y 451.092,Z 277.128,A -85,B 0,C 180,E1 -8848.624,E2 -8848.624} C_VEL
LIN {X 0,Y 450.038,Z 366.016,A -85,B 0,C 180,E1 -8850.135,E2 -8850.135} C_VEL
LIN {X 0,Y 449.639,Z 379.959,A -85,B 0,C 180,E1 -8850.566,E2 -8850.566} C_VEL
LIN {X 0,Y 449.262,Z 392.339,A -85,B 0,C 180,E1 -8851.136,E2 -8851.136} C_VEL
LIN {X 0,Y 448.663,Z 404.669,A -85,B 0,C 180,E1 -8851.906,E2 -8851.906} C_VEL
LIN {X 0,Y 448.101,Z 415.223,A -85,B 0,C 180,E1 -8852.748,E2 -8852.748} C_VEL
LIN {X 0,Y 447.508,Z 425.647,A -85,B 0,C 180,E1 -8853.78,E2 -8853.78} C_VEL
LIN {X 0,Y 446.898,Z 435.201,A -85,B 0,C 180,E1 -8854.957,E2 -8854.957} C_VEL
LIN {X 0,Y 446.372,Z 444.206,A -85,B 0,C 180,E1 -8856.335,E2 -8856.335} C_VEL
LIN {X 0,Y 446.048,Z 450.972,A -85,B 0,C 180,E1 -8857.619,E2 -8857.619} C_VEL
LIN {X 0,Y 445.707,Z 457.166,A -85,B 0,C 180,E1 -8859.093,E2 -8859.093} C_VEL
LIN {X 0,Y 445.503,Z 462.523,A -85,B 0,C 180,E1 -8860.784,E2 -8860.784} C_VEL
LIN {X 0,Y 445.351,Z 465.614,A -85,B 0,C 180,E1 -8862.127,E2 -8862.127} C_VEL
LIN {X 0,Y 445.249,Z 468.328,A -85,B 0,C 180,E1 -8863.976,E2 -8863.976} C_VEL
LIN {X 0,Y 445.226,Z 469.206,A -85,B 0,C 180,E1 -8865.25,E2 -8865.25} C_VEL
LIN {X 0,Y 445.197,Z 469.251,A -85,B 0,C 180,E1 -8866.553,E2 -8866.553} C_VEL
LIN {X 0,Y 445.224,Z 468.448,A -85,B 0,C 180,E1 -8867.881,E2 -8867.881} C_VEL
LIN {X 0,Y 445.31,Z 465.986,A -85,B 0,C 180,E1 -8869.681,E2 -8869.681} C_VEL
LIN {X 0,Y 445.499,Z 461.847,A -85,B 0,C 180,E1 -8871.457,E2 -8871.457} C_VEL
LIN {X 0,Y 445.763,Z 456.033,A -85,B 0,C 180,E1 -8873.196,E2 -8873.196} C_VEL
LIN {X 0,Y 446.071,Z 449.387,A -85,B 0,C 180,E1 -8874.693,E2 -8874.693} C_VEL
LIN {X 0,Y 446.47,Z 441.973,A -85,B 0,C 180,E1 -8876.026,E2 -8876.026} C_VEL
LIN {X 0,Y 446.927,Z 433.326,A -85,B 0,C 180,E1 -8877.281,E2 -8877.281} C_VEL
LIN {X 0,Y 447.459,Z 423.753,A -85,B 0,C 180,E1 -8878.407,E2 -8878.407} C_VEL
LIN {X 0,Y 448.042,Z 412.798,A -85,B 0,C 180,E1 -8879.449,E2 -8879.449} C_VEL
LIN {X 0,Y 448.6,Z 401.433,A -85,B 0,C 180,E1 -8880.303,E2 -8880.303} C_VEL
LIN {X 0,Y 449.137,Z 389.661,A -85,B 0,C 180,E1 -8880.984,E2 -8880.984} C_VEL
LIN {X 0,Y 449.564,Z 377.037,A -85,B 0,C 180,E1 -8881.525,E2 -8881.525} C_VEL
LIN {X 0,Y 449.645,Z 373.893,A -85,B 0,C 180,E1 -8881.63,E2 -8881.63} C_VEL
LIN {X 0,Y 449.02,Z 368.19,A -85,B 0,C 180,E1 -8881.821,E2 -8881.821} C_VEL
LIN {X 0,Y 443.752,Z 349.539,A -85,B 0,C 180,E1 -8882.363,E2 -8882.363} C_VEL
LIN {X 0,Y 443.227,Z 343.73,A -85,B 0,C 180,E1 -8882.479,E2 -8882.479} C_VEL
LIN {X 0,Y 443.814,Z 276.403,A -85,B 0,C 180,E1 -8883.622,E2 -8883.622} C_VEL
LIN {X 0,Y 440.64,Z 258.613,A -85,B 0,C 180,E1 -8884.082,E2 -8884.082} C_VEL
LIN {X 0,Y 441.366,Z 244.751,A -85,B 0,C 180,E1 -8887.041,E2 -8887.041} C_VEL
LIN {X 0,Y 441.148,Z 241.521,A -85,B 0,C 180,E1 -8887.77,E2 -8887.77} C_VEL
LIN {X 0,Y 439.398,Z 232.326,A -85,B 0,C 180,E1 -8889.98,E2 -8889.98} C_VEL
LIN {X 0,Y 439.384,Z 232.25,A -85,B 0,C 180,E1 -8893.645,E2 -8893.645} C_VEL
LIN {X 0,Y 439.388,Z 232.251,A -85,B 0,C 180,E1 -8896.12,E2 -8896.12} C_VEL
LIN {X 0,Y 439.386,Z 232.252,A -85,B 0,C 180,E1 -8898.936,E2 -8898.936} C_VEL
LIN {X 0,Y 439.544,Z 232.232,A -85,B 0,C 180,E1 -8902.377,E2 -8902.377} C_VEL
LIN {X 0,Y 439.552,Z 232.231,A -85,B 0,C 180,E1 -8904.497,E2 -8904.497} C_VEL
LIN {X 0,Y 439.591,Z 232.226,A -85,B 0,C 180,E1 -8907.252,E2 -8907.252} C_VEL
LIN {X 0,Y 439.687,Z 232.21,A -85,B 0,C 180,E1 -8910.002,E2 -8910.002} C_VEL
LIN {X 0,Y 439.592,Z 232.226,A -85,B 0,C 180,E1 -8912.751,E2 -8912.751} C_VEL
LIN {X 0,Y 439.548,Z 232.228,A -85,B 0,C 180,E1 -8916.428,E2 -8916.428} C_VEL
LIN {X 0,Y 439.433,Z 232.249,A -85,B 0,C 180,E1 -8919.204,E2 -8919.204} C_VEL
LIN {X 0,Y 439.434,Z 232.243,A -85,B 0,C 180,E1 -8922.73,E2 -8922.73} C_VEL
LIN {X 0,Y 439.378,Z 232.249,A -85,B 0,C 180,E1 -8926.352,E2 -8926.352} C_VEL
LIN {X 0,Y 439.335,Z 232.262,A -85,B 0,C 180,E1 -8929.631,E2 -8929.631} C_VEL
LIN {X 0,Y 439.3,Z 232.259,A -85,B 0,C 180,E1 -8932.58,E2 -8932.58} C_VEL
LIN {X 0,Y 439.35,Z 232.257,A -85,B 0,C 180,E1 -8935.59,E2 -8935.59} C_VEL
LIN {X 0,Y 439.366,Z 232.251,A -85,B 0,C 180,E1 -8938.678,E2 -8938.678} C_VEL
LIN {X 0,Y 439.327,Z 232.263,A -85,B 0,C 180,E1 -8942.039,E2 -8942.039} C_VEL
LIN {X 0,Y 439.342,Z 232.254,A -85,B 0,C 180,E1 -8945.347,E2 -8945.347} C_VEL
LIN {X 0,Y 439.345,Z 232.258,A -85,B 0,C 180,E1 -8948.6,E2 -8948.6} C_VEL
LIN {X 0,Y 439.358,Z 232.252,A -85,B 0,C 180,E1 -8951.266,E2 -8951.266} C_VEL
LIN {X 0,Y 439.366,Z 232.256,A -85,B 0,C 180,E1 -8954.735,E2 -8954.735} C_VEL
LIN {X 0,Y 439.373,Z 232.25,A -85,B 0,C 180,E1 -8957.805,E2 -8957.805} C_VEL
LIN {X 0,Y 439.415,Z 232.247,A -85,B 0,C 180,E1 -8960.237,E2 -8960.237} C_VEL
LIN {X 0,Y 439.344,Z 232.253,A -85,B 0,C 180,E1 -8963.72,E2 -8963.72} C_VEL
LIN {X 0,Y 439.344,Z 232.26,A -85,B 0,C 180,E1 -8967.061,E2 -8967.061} C_VEL
LIN {X 0,Y 439.356,Z 232.252,A -85,B 0,C 180,E1 -8970.281,E2 -8970.281} C_VEL
LIN {X 0,Y 439.407,Z 232.25,A -85,B 0,C 180,E1 -8973.404,E2 -8973.404} C_VEL
LIN {X 0,Y 439.368,Z 232.25,A -85,B 0,C 180,E1 -8976.437,E2 -8976.437} C_VEL
LIN {X 0,Y 439.374,Z 232.258,A -85,B 0,C 180,E1 -8979.404,E2 -8979.404} C_VEL
LIN {X 0,Y 439.394,Z 232.247,A -85,B 0,C 180,E1 -8982.316,E2 -8982.316} C_VEL
LIN {X 0,Y 439.438,Z 232.245,A -85,B 0,C 180,E1 -8985.181,E2 -8985.181} C_VEL
LIN {X 0,Y 439.478,Z 232.24,A -85,B 0,C 180,E1 -8988.008,E2 -8988.008} C_VEL
LIN {X 0,Y 439.502,Z 232.241,A -85,B 0,C 180,E1 -8991.732,E2 -8991.732} C_VEL
LIN {X 0,Y 439.603,Z 232.222,A -85,B 0,C 180,E1 -8994.502,E2 -8994.502} C_VEL
LIN {X 0,Y 439.635,Z 232.223,A -85,B 0,C 180,E1 -8998.174,E2 -8998.174} C_VEL
LIN {X 0,Y 439.581,Z 232.224,A -85,B 0,C 180,E1 -9000.922,E2 -9000.922} C_VEL
LIN {X 0,Y 439.611,Z 232.221,A -85,B 0,C 180,E1 -9002.755,E2 -9002.755} C_VEL
LIN {X 0,Y 439.569,Z 232.232,A -85,B 0,C 180,E1 -9006.432,E2 -9006.432} C_VEL
LIN {X 0,Y 439.49,Z 232.235,A -85,B 0,C 180,E1 -9009.207,E2 -9009.207} C_VEL
LIN {X 0,Y 439.48,Z 232.239,A -85,B 0,C 180,E1 -9012.942,E2 -9012.942} C_VEL
LIN {X 0,Y 439.462,Z 232.243,A -85,B 0,C 180,E1 -9016.352,E2 -9016.352} C_VEL
LIN {X 0,Y 439.419,Z 232.244,A -85,B 0,C 180,E1 -9019.63,E2 -9019.63} C_VEL
LIN {X 0,Y 439.38,Z 232.254,A -85,B 0,C 180,E1 -9022.579,E2 -9022.579} C_VEL
LIN {X 0,Y 439.389,Z 232.249,A -85,B 0,C 180,E1 -9025.591,E2 -9025.591} C_VEL
LIN {X 0,Y 439.402,Z 232.25,A -85,B 0,C 180,E1 -9028.679,E2 -9028.679} C_VEL
LIN {X 0,Y 439.383,Z 232.248,A -85,B 0,C 180,E1 -9032.031,E2 -9032.031} C_VEL
LIN {X 0,Y 439.41,Z 232.253,A -85,B 0,C 180,E1 -9035.342,E2 -9035.342} C_VEL
LIN {X 0,Y 439.382,Z 232.249,A -85,B 0,C 180,E1 -9038.6,E2 -9038.6} C_VEL
LIN {X 0,Y 439.367,Z 232.251,A -85,B 0,C 180,E1 -9042.212,E2 -9042.212} C_VEL
LIN {X 0,Y 439.39,Z 232.251,A -85,B 0,C 180,E1 -9045.268,E2 -9045.268} C_VEL
LIN {X 0,Y 439.373,Z 232.25,A -85,B 0,C 180,E1 -9049.017,E2 -9049.017} C_VEL
LIN {X 0,Y 439.377,Z 232.255,A -85,B 0,C 180,E1 -9051.612,E2 -9051.612} C_VEL
LIN {X 0,Y 439.413,Z 232.245,A -85,B 0,C 180,E1 -9054.844,E2 -9054.844} C_VEL
LIN {X 0,Y 439.389,Z 232.256,A -85,B 0,C 180,E1 -9058.14,E2 -9058.14} C_VEL
LIN {X 0,Y 439.424,Z 232.249,A -85,B 0,C 180,E1 -9061.606,E2 -9061.606} C_VEL
LIN {X 0,Y 439.485,Z 232.391,A -85,B 0,C 180,E1 -9064.238,E2 -9064.238} C_VEL
LIN {X 0,Y 441.669,Z 243.95,A -85,B 0,C 180,E1 -9066.779,E2 -9066.779} C_VEL
LIN {X 0,Y 441.692,Z 248.903,A -85,B 0,C 180,E1 -9067.795,E2 -9067.795} C_VEL
LIN {X 0,Y 440.676,Z 266.926,A -85,B 0,C 180,E1 -9071.398,E2 -9071.398} C_VEL
LIN {X 0,Y 440.516,Z 269.764,A -85,B 0,C 180,E1 -9071.921,E2 -9071.921} C_VEL
LIN {X 0,Y 441.195,Z 274.157,A -85,B 0,C 180,E1 -9072.076,E2 -9072.076} C_VEL
LIN {X 0,Y 443.924,Z 291.943,A -85,B 0,C 180,E1 -9072.493,E2 -9072.493} C_VEL
LIN {X 0,Y 442.964,Z 378.188,A -85,B 0,C 180,E1 -9073.967,E2 -9073.967} C_VEL
LIN {X 0,Y 442.543,Z 391.885,A -85,B 0,C 180,E1 -9074.395,E2 -9074.395} C_VEL
LIN {X 0,Y 442.03,Z 404.263,A -85,B 0,C 180,E1 -9074.967,E2 -9074.967} C_VEL
LIN {X 0,Y 441.415,Z 416.143,A -85,B 0,C 180,E1 -9075.711,E2 -9075.711} C_VEL
LIN {X 0,Y 440.815,Z 427.886,A -85,B 0,C 180,E1 -9076.66,E2 -9076.66} C_VEL
LIN {X 0,Y 440.275,Z 437.897,A -85,B 0,C 180,E1 -9077.671,E2 -9077.671} C_VEL
LIN {X 0,Y 439.603,Z 447.97,A -85,B 0,C 180,E1 -9078.938,E2 -9078.938} C_VEL
LIN {X 0,Y 439.113,Z 456.835,A -85,B 0,C 180,E1 -9080.324,E2 -9080.324} C_VEL
LIN {X 0,Y 438.793,Z 463.912,A -85,B 0,C 180,E1 -9081.71,E2 -9081.71} C_VEL
LIN {X 0,Y 438.527,Z 469.561,A -85,B 0,C 180,E1 -9083.095,E2 -9083.095} C_VEL
LIN {X 0,Y 438.411,Z 473.997,A -85,B 0,C 180,E1 -9084.479,E2 -9084.479} C_VEL
LIN {X 0,Y 438.35,Z 476.337,A -85,B 0,C 180,E1 -9085.4,E2 -9085.4} C_VEL
LIN {X 0,Y 438.264,Z 478.243,A -85,B 0,C 180,E1 -9086.321,E2 -9086.321} C_VEL
LIN {X 0,Y 438.299,Z 479.69,A -85,B 0,C 180,E1 -9087.241,E2 -9087.241} C_VEL
LIN {X 0,Y 438.279,Z 480.71,A -85,B 0,C 180,E1 -9088.161,E2 -9088.161} C_VEL
LIN {X 0,Y 438.234,Z 481.576,A -85,B 0,C 180,E1 -9089.998,E2 -9089.998} C_VEL
LIN {X 0,Y 438.236,Z 481.38,A -85,B 0,C 180,E1 -9090.917,E2 -9090.917} C_VEL
LIN {X 0,Y 438.279,Z 480.777,A -85,B 0,C 180,E1 -9091.836,E2 -9091.836} C_VEL
LIN {X 0,Y 438.298,Z 479.783,A -85,B 0,C 180,E1 -9092.756,E2 -9092.756} C_VEL
LIN {X 0,Y 438.263,Z 478.388,A -85,B 0,C 180,E1 -9093.676,E2 -9093.676} C_VEL
LIN {X 0,Y 438.424,Z 475.445,A -85,B 0,C 180,E1 -9095.056,E2 -9095.056} C_VEL
LIN {X 0,Y 438.478,Z 471.457,A -85,B 0,C 180,E1 -9096.44,E2 -9096.44} C_VEL
LIN {X 0,Y 438.746,Z 465.324,A -85,B 0,C 180,E1 -9098.055,E2 -9098.055} C_VEL
LIN {X 0,Y 439.092,Z 458.616,A -85,B 0,C 180,E1 -9099.441,E2 -9099.441} C_VEL
LIN {X 0,Y 439.551,Z 450.29,A -85,B 0,C 180,E1 -9100.827,E2 -9100.827} C_VEL
LIN {X 0,Y 440.144,Z 441.753,A -85,B 0,C 180,E1 -9101.979,E2 -9101.979} C_VEL
LIN {X 0,Y 440.843,Z 431.073,A -85,B 0,C 180,E1 -9103.142,E2 -9103.142} C_VEL
LIN {X 0,Y 441.333,Z 420.777,A -85,B 0,C 180,E1 -9104.053,E2 -9104.053} C_VEL
LIN {X 0,Y 441.969,Z 409.342,A -85,B 0,C 180,E1 -9104.855,E2 -9104.855} C_VEL
LIN {X 0,Y 442.54,Z 397.565,A -85,B 0,C 180,E1 -9105.484,E2 -9105.484} C_VEL
LIN {X 0,Y 443.046,Z 384.072,A -85,B 0,C 180,E1 -9105.997,E2 -9105.997} C_VEL
LIN {X 0,Y 443.398,Z 370.657,A -85,B 0,C 180,E1 -9106.309,E2 -9106.309} C_VEL
LIN {X 0,Y 444.21,Z 290.354,A -85,B 0,C 180,E1 -9107.688,E2 -9107.688} C_VEL
LIN {X 0,Y 440.64,Z 269.367,A -85,B 0,C 180,E1 -9108.25,E2 -9108.25} C_VEL
LIN {X 0,Y 441.369,Z 253.787,A -85,B 0,C 180,E1 -9111.237,E2 -9111.237} C_VEL
LIN {X 0,Y 441.782,Z 244.914,A -85,B 0,C 180,E1 -9112.984,E2 -9112.984} C_VEL
LIN {X 0,Y 439.762,Z 234.004,A -85,B 0,C 180,E1 -9115.307,E2 -9115.307} C_VEL
LIN {X 0,Y 439.431,Z 232.28,A -85,B 0,C 180,E1 -9115.762,E2 -9115.762} C_VEL
LIN {X 0,Y 439.425,Z 232.248,A -85,B 0,C 180,E1 -9118.671,E2 -9118.671} C_VEL
LIN {X 0,Y 439.377,Z 232.257,A -85,B 0,C 180,E1 -9122.027,E2 -9122.027} C_VEL
LIN {X 0,Y 439.399,Z 232.251,A -85,B 0,C 180,E1 -9125.336,E2 -9125.336} C_VEL
LIN {X 0,Y 439.367,Z 232.254,A -85,B 0,C 180,E1 -9128.594,E2 -9128.594} C_VEL
LIN {X 0,Y 439.355,Z 232.259,A -85,B 0,C 180,E1 -9132.206,E2 -9132.206} C_VEL
LIN {X 0,Y 439.379,Z 232.25,A -85,B 0,C 180,E1 -9135.263,E2 -9135.263} C_VEL
LIN {X 0,Y 439.365,Z 232.255,A -85,B 0,C 180,E1 -9138.743,E2 -9138.743} C_VEL
LIN {X 0,Y 439.357,Z 232.253,A -85,B 0,C 180,E1 -9141.607,E2 -9141.607} C_VEL
LIN {X 0,Y 439.391,Z 232.252,A -85,B 0,C 180,E1 -9144.839,E2 -9144.839} C_VEL
LIN {X 0,Y 439.369,Z 232.254,A -85,B 0,C 180,E1 -9148.135,E2 -9148.135} C_VEL
LIN {X 0,Y 439.385,Z 232.25,A -85,B 0,C 180,E1 -9151.605,E2 -9151.605} C_VEL
LIN {X 0,Y 439.362,Z 232.252,A -85,B 0,C 180,E1 -9154.408,E2 -9154.408} C_VEL
LIN {X 0,Y 439.349,Z 232.252,A -85,B 0,C 180,E1 -9157.419,E2 -9157.419} C_VEL
LIN {X 0,Y 439.38,Z 232.252,A -85,B 0,C 180,E1 -9160.679,E2 -9160.679} C_VEL
LIN {X 0,Y 439.407,Z 232.246,A -85,B 0,C 180,E1 -9164.217,E2 -9164.217} C_VEL
LIN {X 0,Y 439.476,Z 232.238,A -85,B 0,C 180,E1 -9167.28,E2 -9167.28} C_VEL
LIN {X 0,Y 439.47,Z 232.243,A -85,B 0,C 180,E1 -9170.792,E2 -9170.792} C_VEL
LIN {X 0,Y 439.58,Z 232.225,A -85,B 0,C 180,E1 -9173.569,E2 -9173.569} C_VEL
LIN {X 0,Y 439.595,Z 232.227,A -85,B 0,C 180,E1 -9177.245,E2 -9177.245} C_VEL
LIN {X 0,Y 439.74,Z 232.204,A -85,B 0,C 180,E1 -9179.994,E2 -9179.994} C_VEL
LIN {X 0,Y 439.619,Z 232.221,A -85,B 0,C 180,E1 -9182.743,E2 -9182.743} C_VEL
LIN {X 0,Y 439.563,Z 232.228,A -85,B 0,C 180,E1 -9186.474,E2 -9186.474} C_VEL
LIN {X 0,Y 439.476,Z 232.243,A -85,B 0,C 180,E1 -9189.195,E2 -9189.195} C_VEL
LIN {X 0,Y 439.476,Z 232.24,A -85,B 0,C 180,E1 -9192.72,E2 -9192.72} C_VEL
LIN {X 0,Y 439.416,Z 232.249,A -85,B 0,C 180,E1 -9196.343,E2 -9196.343} C_VEL
LIN {X 0,Y 439.401,Z 232.252,A -85,B 0,C 180,E1 -9199.619,E2 -9199.619} C_VEL
LIN {X 0,Y 439.401,Z 232.329,A -85,B 0,C 180,E1 -9202.689,E2 -9202.689} C_VEL
LIN {X 0,Y 440.428,Z 237.07,A -85,B 0,C 180,E1 -9203.752,E2 -9203.752} C_VEL
LIN {X 0,Y 441.311,Z 242.217,A -85,B 0,C 180,E1 -9204.81,E2 -9204.81} C_VEL
LIN {X 0,Y 440.719,Z 257.941,A -85,B 0,C 180,E1 -9207.795,E2 -9207.795} C_VEL
LIN {X 0,Y 444.273,Z 276.932,A -85,B 0,C 180,E1 -9208.323,E2 -9208.323} C_VEL
LIN {X 0,Y 443.236,Z 366.683,A -85,B 0,C 180,E1 -9209.89,E2 -9209.89} C_VEL
LIN {X 0,Y 442.828,Z 380.105,A -85,B 0,C 180,E1 -9210.315,E2 -9210.315} C_VEL
LIN {X 0,Y 442.439,Z 391.477,A -85,B 0,C 180,E1 -9210.84,E2 -9210.84} C_VEL
LIN {X 0,Y 441.873,Z 403.131,A -85,B 0,C 180,E1 -9211.554,E2 -9211.554} C_VEL
LIN {X 0,Y 441.291,Z 414.23,A -85,B 0,C 180,E1 -9212.431,E2 -9212.431} C_VEL
LIN {X 0,Y 440.589,Z 425.146,A -85,B 0,C 180,E1 -9213.509,E2 -9213.509} C_VEL
LIN {X 0,Y 439.991,Z 434.614,A -85,B 0,C 180,E1 -9214.673,E2 -9214.673} C_VEL
LIN {X 0,Y 439.403,Z 443.558,A -85,B 0,C 180,E1 -9216.041,E2 -9216.041} C_VEL
LIN {X 0,Y 439.022,Z 451,A -85,B 0,C 180,E1 -9217.457,E2 -9217.457} C_VEL
LIN {X 0,Y 438.733,Z 456.068,A -85,B 0,C 180,E1 -9218.652,E2 -9218.652} C_VEL
LIN {X 0,Y 438.514,Z 460.256,A -85,B 0,C 180,E1 -9219.861,E2 -9219.861} C_VEL
LIN {X 0,Y 438.364,Z 463.687,A -85,B 0,C 180,E1 -9221.107,E2 -9221.107} C_VEL
LIN {X 0,Y 438.253,Z 466.48,A -85,B 0,C 180,E1 -9222.47,E2 -9222.47} C_VEL
LIN {X 0,Y 438.162,Z 468.311,A -85,B 0,C 180,E1 -9223.801,E2 -9223.801} C_VEL
LIN {X 0,Y 438.141,Z 469.248,A -85,B 0,C 180,E1 -9225.11,E2 -9225.11} C_VEL
LIN {X 0,Y 438.105,Z 469.379,A -85,B 0,C 180,E1 -9226.389,E2 -9226.389} C_VEL
LIN {X 0,Y 438.134,Z 468.766,A -85,B 0,C 180,E1 -9227.649,E2 -9227.649} C_VEL
LIN {X 0,Y 438.19,Z 467.4,A -85,B 0,C 180,E1 -9228.908,E2 -9228.908} C_VEL
LIN {X 0,Y 438.263,Z 464.928,A -85,B 0,C 180,E1 -9230.315,E2 -9230.315} C_VEL
LIN {X 0,Y 438.429,Z 461.343,A -85,B 0,C 180,E1 -9231.749,E2 -9231.749} C_VEL
LIN {X 0,Y 438.676,Z 456.443,A -85,B 0,C 180,E1 -9233.215,E2 -9233.215} C_VEL
LIN {X 0,Y 439.031,Z 449.488,A -85,B 0,C 180,E1 -9234.813,E2 -9234.813} C_VEL
LIN {X 0,Y 439.453,Z 441.581,A -85,B 0,C 180,E1 -9236.248,E2 -9236.248} C_VEL
LIN {X 0,Y 439.959,Z 433.08,A -85,B 0,C 180,E1 -9237.484,E2 -9237.484} C_VEL
LIN {X 0,Y 440.509,Z 423.362,A -85,B 0,C 180,E1 -9238.636,E2 -9238.636} C_VEL
LIN {X 0,Y 441.068,Z 413.242,A -85,B 0,C 180,E1 -9239.611,E2 -9239.611} C_VEL
LIN {X 0,Y 441.681,Z 401.402,A -85,B 0,C 180,E1 -9240.516,E2 -9240.516} C_VEL
LIN {X 0,Y 442.277,Z 389.038,A -85,B 0,C 180,E1 -9241.237,E2 -9241.237} C_VEL
LIN {X 0,Y 442.697,Z 376.143,A -85,B 0,C 180,E1 -9241.787,E2 -9241.787} C_VEL
LIN {X 0,Y 443.01,Z 362.896,A -85,B 0,C 180,E1 -9242.147,E2 -9242.147} C_VEL
LIN {X 0,Y 443.227,Z 343.73,A -85,B 0,C 180,E1 -9242.479,E2 -9242.479} C_VEL
LIN {X 0,Y 442.69,Z 337.925,A -85,B 0,C 180,E1 -9242.599,E2 -9242.599} C_VEL
LIN {X 0,Y 437.408,Z 319.224,A -85,B 0,C 180,E1 -9243.115,E2 -9243.115} C_VEL
LIN {X 0,Y 436.752,Z 313.421,A -85,B 0,C 180,E1 -9243.241,E2 -9243.241} C_VEL
LIN {X 0,Y 437.128,Z 277.952,A -85,B 0,C 180,E1 -9243.858,E2 -9243.858} C_VEL
LIN {X 0,Y 433.719,Z 258.973,A -85,B 0,C 180,E1 -9244.347,E2 -9244.347} C_VEL
LIN {X 0,Y 433.724,Z 257.508,A -85,B 0,C 180,E1 -9244.573,E2 -9244.573} C_VEL
LIN {X 0,Y 434.42,Z 244.947,A -85,B 0,C 180,E1 -9247.346,E2 -9247.346} C_VEL
LIN {X 0,Y 433.186,Z 237.561,A -85,B 0,C 180,E1 -9249.09,E2 -9249.09} C_VEL
LIN {X 0,Y 432.35,Z 233.171,A -85,B 0,C 180,E1 -9250.203,E2 -9250.203} C_VEL
LIN {X 0,Y 432.37,Z 233.126,A -85,B 0,C 180,E1 -9253.961,E2 -9253.961} C_VEL
LIN {X 0,Y 432.41,Z 233.117,A -85,B 0,C 180,E1 -9257.804,E2 -9257.804} C_VEL
LIN {X 0,Y 432.417,Z 233.116,A -85,B 0,C 180,E1 -9261.591,E2 -9261.591} C_VEL
LIN {X 0,Y 432.528,Z 233.105,A -85,B 0,C 180,E1 -9264.407,E2 -9264.407} C_VEL
LIN {X 0,Y 432.532,Z 233.102,A -85,B 0,C 180,E1 -9268.139,E2 -9268.139} C_VEL
LIN {X 0,Y 432.658,Z 233.086,A -85,B 0,C 180,E1 -9270.002,E2 -9270.002} C_VEL
LIN {X 0,Y 432.542,Z 233.105,A -85,B 0,C 180,E1 -9272.796,E2 -9272.796} C_VEL
LIN {X 0,Y 432.502,Z 233.106,A -85,B 0,C 180,E1 -9276.533,E2 -9276.533} C_VEL
LIN {X 0,Y 432.377,Z 233.129,A -85,B 0,C 180,E1 -9279.356,E2 -9279.356} C_VEL
LIN {X 0,Y 432.375,Z 233.123,A -85,B 0,C 180,E1 -9282.816,E2 -9282.816} C_VEL
LIN {X 0,Y 432.343,Z 233.125,A -85,B 0,C 180,E1 -9286.483,E2 -9286.483} C_VEL
LIN {X 0,Y 432.271,Z 233.139,A -85,B 0,C 180,E1 -9289.965,E2 -9289.965} C_VEL
LIN {X 0,Y 432.255,Z 233.137,A -85,B 0,C 180,E1 -9292.969,E2 -9292.969} C_VEL
LIN {X 0,Y 432.307,Z 233.136,A -85,B 0,C 180,E1 -9296.038,E2 -9296.038} C_VEL
LIN {X 0,Y 432.293,Z 233.132,A -85,B 0,C 180,E1 -9299.192,E2 -9299.192} C_VEL
LIN {X 0,Y 432.276,Z 233.139,A -85,B 0,C 180,E1 -9302.301,E2 -9302.301} C_VEL
LIN {X 0,Y 432.286,Z 233.135,A -85,B 0,C 180,E1 -9304.683,E2 -9304.683} C_VEL
LIN {X 0,Y 432.3,Z 233.137,A -85,B 0,C 180,E1 -9308.155,E2 -9308.155} C_VEL
LIN {X 0,Y 432.327,Z 233.128,A -85,B 0,C 180,E1 -9311.615,E2 -9311.615} C_VEL
LIN {X 0,Y 432.336,Z 233.132,A -85,B 0,C 180,E1 -9314.348,E2 -9314.348} C_VEL
LIN {X 0,Y 432.326,Z 233.13,A -85,B 0,C 180,E1 -9317.016,E2 -9317.016} C_VEL
LIN {X 0,Y 432.321,Z 233.128,A -85,B 0,C 180,E1 -9319.824,E2 -9319.824} C_VEL
LIN {X 0,Y 432.283,Z 233.138,A -85,B 0,C 180,E1 -9323.03,E2 -9323.03} C_VEL
LIN {X 0,Y 432.329,Z 233.127,A -85,B 0,C 180,E1 -9326.004,E2 -9326.004} C_VEL
LIN {X 0,Y 432.321,Z 233.13,A -85,B 0,C 180,E1 -9329.497,E2 -9329.497} C_VEL
LIN {X 0,Y 432.369,Z 233.128,A -85,B 0,C 180,E1 -9332.936,E2 -9332.936} C_VEL
LIN {X 0,Y 432.352,Z 233.125,A -85,B 0,C 180,E1 -9336.031,E2 -9336.031} C_VEL
LIN {X 0,Y 432.336,Z 233.131,A -85,B 0,C 180,E1 -9339.053,E2 -9339.053} C_VEL
LIN {X 0,Y 432.349,Z 233.126,A -85,B 0,C 180,E1 -9342.018,E2 -9342.018} C_VEL
LIN {X 0,Y 432.386,Z 233.121,A -85,B 0,C 180,E1 -9344.934,E2 -9344.934} C_VEL
LIN {X 0,Y 432.454,Z 233.118,A -85,B 0,C 180,E1 -9347.81,E2 -9347.81} C_VEL
LIN {X 0,Y 432.462,Z 233.116,A -85,B 0,C 180,E1 -9351.597,E2 -9351.597} C_VEL
LIN {X 0,Y 432.577,Z 233.098,A -85,B 0,C 180,E1 -9354.412,E2 -9354.412} C_VEL
LIN {X 0,Y 432.605,Z 233.099,A -85,B 0,C 180,E1 -9358.144,E2 -9358.144} C_VEL
LIN {X 0,Y 432.543,Z 233.101,A -85,B 0,C 180,E1 -9360.937,E2 -9360.937} C_VEL
LIN {X 0,Y 432.565,Z 233.099,A -85,B 0,C 180,E1 -9362.8,E2 -9362.8} C_VEL
LIN {X 0,Y 432.582,Z 233.097,A -85,B 0,C 180,E1 -9365.6,E2 -9365.6} C_VEL
LIN {X 0,Y 432.459,Z 233.119,A -85,B 0,C 180,E1 -9368.416,E2 -9368.416} C_VEL
LIN {X 0,Y 432.472,Z 233.114,A -85,B 0,C 180,E1 -9372.202,E2 -9372.202} C_VEL
LIN {X 0,Y 432.445,Z 233.114,A -85,B 0,C 180,E1 -9376.044,E2 -9376.044} C_VEL
LIN {X 0,Y 432.404,Z 233.118,A -85,B 0,C 180,E1 -9379.489,E2 -9379.489} C_VEL
LIN {X 0,Y 432.328,Z 233.134,A -85,B 0,C 180,E1 -9382.969,E2 -9382.969} C_VEL
LIN {X 0,Y 432.338,Z 233.126,A -85,B 0,C 180,E1 -9386.039,E2 -9386.039} C_VEL
LIN {X 0,Y 432.342,Z 233.132,A -85,B 0,C 180,E1 -9389.192,E2 -9389.192} C_VEL
LIN {X 0,Y 432.341,Z 233.126,A -85,B 0,C 180,E1 -9392.446,E2 -9392.446} C_VEL
LIN {X 0,Y 432.356,Z 233.125,A -85,B 0,C 180,E1 -9395.821,E2 -9395.821} C_VEL
LIN {X 0,Y 432.323,Z 233.136,A -85,B 0,C 180,E1 -9399.35,E2 -9399.35} C_VEL
LIN {X 0,Y 432.323,Z 233.132,A -85,B 0,C 180,E1 -9401.803,E2 -9401.803} C_VEL
LIN {X 0,Y 432.332,Z 233.127,A -85,B 0,C 180,E1 -9404.352,E2 -9404.352} C_VEL
LIN {X 0,Y 432.302,Z 233.132,A -85,B 0,C 180,E1 -9407.023,E2 -9407.023} C_VEL
LIN {X 0,Y 432.309,Z 233.137,A -85,B 0,C 180,E1 -9409.829,E2 -9409.829} C_VEL
LIN {X 0,Y 432.318,Z 233.129,A -85,B 0,C 180,E1 -9413.022,E2 -9413.022} C_VEL
LIN {X 0,Y 432.364,Z 233.131,A -85,B 0,C 180,E1 -9416.001,E2 -9416.001} C_VEL
LIN {X 0,Y 432.362,Z 233.124,A -85,B 0,C 180,E1 -9419.492,E2 -9419.492} C_VEL
LIN {X 0,Y 432.364,Z 233.131,A -85,B 0,C 180,E1 -9421.874,E2 -9421.874} C_VEL
LIN {X 0,Y 432.438,Z 233.331,A -85,B 0,C 180,E1 -9424.036,E2 -9424.036} C_VEL
LIN {X 0,Y 434.683,Z 245.095,A -85,B 0,C 180,E1 -9426.663,E2 -9426.663} C_VEL
LIN {X 0,Y 434.822,Z 248.722,A -85,B 0,C 180,E1 -9427.425,E2 -9427.425} C_VEL
LIN {X 0,Y 433.731,Z 266.754,A -85,B 0,C 180,E1 -9431.089,E2 -9431.089} C_VEL
LIN {X 0,Y 433.595,Z 269.738,A -85,B 0,C 180,E1 -9431.65,E2 -9431.65} C_VEL
LIN {X 0,Y 434.394,Z 274.985,A -85,B 0,C 180,E1 -9431.82,E2 -9431.82} C_VEL
LIN {X 0,Y 437.113,Z 292.42,A -85,B 0,C 180,E1 -9432.239,E2 -9432.239} C_VEL
LIN {X 0,Y 436.086,Z 378.371,A -85,B 0,C 180,E1 -9433.737,E2 -9433.737} C_VEL
LIN {X 0,Y 435.669,Z 391.968,A -85,B 0,C 180,E1 -9434.172,E2 -9434.172} C_VEL
LIN {X 0,Y 435.103,Z 404.791,A -85,B 0,C 180,E1 -9434.781,E2 -9434.781} C_VEL
LIN {X 0,Y 434.444,Z 417.329,A -85,B 0,C 180,E1 -9435.597,E2 -9435.597} C_VEL
LIN {X 0,Y 433.826,Z 428.378,A -85,B 0,C 180,E1 -9436.518,E2 -9436.518} C_VEL
LIN {X 0,Y 433.237,Z 438.605,A -85,B 0,C 180,E1 -9437.586,E2 -9437.586} C_VEL
LIN {X 0,Y 432.618,Z 447.72,A -85,B 0,C 180,E1 -9438.757,E2 -9438.757} C_VEL
LIN {X 0,Y 432.092,Z 456.614,A -85,B 0,C 180,E1 -9440.165,E2 -9440.165} C_VEL
LIN {X 0,Y 431.731,Z 463.725,A -85,B 0,C 180,E1 -9441.574,E2 -9441.574} C_VEL
LIN {X 0,Y 431.45,Z 469.394,A -85,B 0,C 180,E1 -9442.981,E2 -9442.981} C_VEL
LIN {X 0,Y 431.314,Z 473.847,A -85,B 0,C 180,E1 -9444.388,E2 -9444.388} C_VEL
LIN {X 0,Y 431.281,Z 476.196,A -85,B 0,C 180,E1 -9445.325,E2 -9445.325} C_VEL
LIN {X 0,Y 431.174,Z 478.11,A -85,B 0,C 180,E1 -9446.26,E2 -9446.26} C_VEL
LIN {X 0,Y 431.195,Z 479.57,A -85,B 0,C 180,E1 -9447.196,E2 -9447.196} C_VEL
LIN {X 0,Y 431.203,Z 480.597,A -85,B 0,C 180,E1 -9448.13,E2 -9448.13} C_VEL
LIN {X 0,Y 431.15,Z 481.475,A -85,B 0,C 180,E1 -9449.998,E2 -9449.998} C_VEL
LIN {X 0,Y 431.154,Z 481.289,A -85,B 0,C 180,E1 -9450.932,E2 -9450.932} C_VEL
LIN {X 0,Y 431.203,Z 480.691,A -85,B 0,C 180,E1 -9451.866,E2 -9451.866} C_VEL
LIN {X 0,Y 431.194,Z 479.7,A -85,B 0,C 180,E1 -9452.801,E2 -9452.801} C_VEL
LIN {X 0,Y 431.173,Z 478.309,A -85,B 0,C 180,E1 -9453.737,E2 -9453.737} C_VEL
LIN {X 0,Y 431.336,Z 475.372,A -85,B 0,C 180,E1 -9455.14,E2 -9455.14} C_VEL
LIN {X 0,Y 431.395,Z 471.391,A -85,B 0,C 180,E1 -9456.547,E2 -9456.547} C_VEL
LIN {X 0,Y 431.702,Z 465.269,A -85,B 0,C 180,E1 -9458.188,E2 -9458.188} C_VEL
LIN {X 0,Y 432.08,Z 458.566,A -85,B 0,C 180,E1 -9459.595,E2 -9459.595} C_VEL
LIN {X 0,Y 432.556,Z 450.248,A -85,B 0,C 180,E1 -9461.004,E2 -9461.004} C_VEL
LIN {X 0,Y 433.185,Z 441.723,A -85,B 0,C 180,E1 -9462.174,E2 -9462.174} C_VEL
LIN {X 0,Y 433.866,Z 431.747,A -85,B 0,C 180,E1 -9463.289,E2 -9463.289} C_VEL
LIN {X 0,Y 434.435,Z 420.807,A -85,B 0,C 180,E1 -9464.281,E2 -9464.281} C_VEL
LIN {X 0,Y 435.117,Z 409.43,A -85,B 0,C 180,E1 -9465.095,E2 -9465.095} C_VEL
LIN {X 0,Y 435.729,Z 397.761,A -85,B 0,C 180,E1 -9465.732,E2 -9465.732} C_VEL
LIN {X 0,Y 436.239,Z 384.429,A -85,B 0,C 180,E1 -9466.253,E2 -9466.253} C_VEL
LIN {X 0,Y 436.619,Z 371.483,A -85,B 0,C 180,E1 -9466.569,E2 -9466.569} C_VEL
LIN {X 0,Y 437.479,Z 290.918,A -85,B 0,C 180,E1 -9467.979,E2 -9467.979} C_VEL
LIN {X 0,Y 433.739,Z 269.402,A -85,B 0,C 180,E1 -9468.564,E2 -9468.564} C_VEL
LIN {X 0,Y 434.007,Z 263.699,A -85,B 0,C 180,E1 -9469.632,E2 -9469.632} C_VEL
LIN {X 0,Y 434.906,Z 247.212,A -85,B 0,C 180,E1 -9472.905,E2 -9472.905} C_VEL
LIN {X 0,Y 433.473,Z 238.494,A -85,B 0,C 180,E1 -9474.772,E2 -9474.772} C_VEL
LIN {X 0,Y 432.421,Z 233.209,A -85,B 0,C 180,E1 -9475.994,E2 -9475.994} C_VEL
LIN {X 0,Y 432.351,Z 233.128,A -85,B 0,C 180,E1 -9479.185,E2 -9479.185} C_VEL
LIN {X 0,Y 432.331,Z 233.133,A -85,B 0,C 180,E1 -9482.44,E2 -9482.44} C_VEL
LIN {X 0,Y 432.35,Z 233.132,A -85,B 0,C 180,E1 -9485.628,E2 -9485.628} C_VEL
LIN {X 0,Y 432.33,Z 233.13,A -85,B 0,C 180,E1 -9488.708,E2 -9488.708} C_VEL
LIN {X 0,Y 432.31,Z 233.134,A -85,B 0,C 180,E1 -9491.797,E2 -9491.797} C_VEL
LIN {X 0,Y 432.337,Z 233.133,A -85,B 0,C 180,E1 -9494.344,E2 -9494.344} C_VEL
LIN {X 0,Y 432.306,Z 233.132,A -85,B 0,C 180,E1 -9497.015,E2 -9497.015} C_VEL
LIN {X 0,Y 432.291,Z 233.137,A -85,B 0,C 180,E1 -9499.824,E2 -9499.824} C_VEL
LIN {X 0,Y 432.297,Z 233.132,A -85,B 0,C 180,E1 -9503.016,E2 -9503.016} C_VEL
LIN {X 0,Y 432.333,Z 233.131,A -85,B 0,C 180,E1 -9505.998,E2 -9505.998} C_VEL
LIN {X 0,Y 432.341,Z 233.126,A -85,B 0,C 180,E1 -9509.487,E2 -9509.487} C_VEL
LIN {X 0,Y 432.318,Z 233.131,A -85,B 0,C 180,E1 -9511.867,E2 -9511.867} C_VEL
LIN {X 0,Y 432.318,Z 233.134,A -85,B 0,C 180,E1 -9514.992,E2 -9514.992} C_VEL
LIN {X 0,Y 432.347,Z 233.124,A -85,B 0,C 180,E1 -9518.04,E2 -9518.04} C_VEL
LIN {X 0,Y 432.337,Z 233.129,A -85,B 0,C 180,E1 -9521.022,E2 -9521.022} C_VEL
LIN {X 0,Y 432.376,Z 233.121,A -85,B 0,C 180,E1 -9523.954,E2 -9523.954} C_VEL
LIN {X 0,Y 432.448,Z 233.11,A -85,B 0,C 180,E1 -9527.798,E2 -9527.798} C_VEL
LIN {X 0,Y 432.437,Z 233.117,A -85,B 0,C 180,E1 -9531.584,E2 -9531.584} C_VEL
LIN {X 0,Y 432.569,Z 233.097,A -85,B 0,C 180,E1 -9534.4,E2 -9534.4} C_VEL
LIN {X 0,Y 432.579,Z 233.098,A -85,B 0,C 180,E1 -9538.132,E2 -9538.132} C_VEL
LIN {X 0,Y 432.71,Z 233.08,A -85,B 0,C 180,E1 -9539.994,E2 -9539.994} C_VEL
LIN {X 0,Y 432.571,Z 233.099,A -85,B 0,C 180,E1 -9542.787,E2 -9542.787} C_VEL
LIN {X 0,Y 432.52,Z 233.106,A -85,B 0,C 180,E1 -9546.476,E2 -9546.476} C_VEL
LIN {X 0,Y 432.419,Z 233.122,A -85,B 0,C 180,E1 -9549.347,E2 -9549.347} C_VEL
LIN {X 0,Y 432.417,Z 233.12,A -85,B 0,C 180,E1 -9552.806,E2 -9552.806} C_VEL
LIN {X 0,Y 432.381,Z 233.125,A -85,B 0,C 180,E1 -9556.473,E2 -9556.473} C_VEL
LIN {X 0,Y 432.348,Z 233.133,A -85,B 0,C 180,E1 -9559.952,E2 -9559.952} C_VEL
LIN {X 0,Y 432.394,Z 233.298,A -85,B 0,C 180,E1 -9562.473,E2 -9562.473} C_VEL
LIN {X 0,Y 434.365,Z 243.22,A -85,B 0,C 180,E1 -9564.614,E2 -9564.614} C_VEL
LIN {X 0,Y 433.836,Z 258.061,A -85,B 0,C 180,E1 -9567.471,E2 -9567.471} C_VEL
LIN {X 0,Y 437.611,Z 278.111,A -85,B 0,C 180,E1 -9568.042,E2 -9568.042} C_VEL
LIN {X 0,Y 436.467,Z 366.306,A -85,B 0,C 180,E1 -9569.603,E2 -9569.603} C_VEL
LIN {X 0,Y 436.025,Z 380.34,A -85,B 0,C 180,E1 -9570.052,E2 -9570.052} C_VEL
LIN {X 0,Y 435.568,Z 393.213,A -85,B 0,C 180,E1 -9570.673,E2 -9570.673} C_VEL
LIN {X 0,Y 434.89,Z 405.627,A -85,B 0,C 180,E1 -9571.484,E2 -9571.484} C_VEL
LIN {X 0,Y 434.226,Z 417.207,A -85,B 0,C 180,E1 -9572.461,E2 -9572.461} C_VEL
LIN {X 0,Y 433.534,Z 427.548,A -85,B 0,C 180,E1 -9573.564,E2 -9573.564} C_VEL
LIN {X 0,Y 432.869,Z 436.679,A -85,B 0,C 180,E1 -9574.76,E2 -9574.76} C_VEL
LIN {X 0,Y 432.341,Z 444.972,A -85,B 0,C 180,E1 -9576.095,E2 -9576.095} C_VEL
LIN {X 0,Y 431.89,Z 452.564,A -85,B 0,C 180,E1 -9577.635,E2 -9577.635} C_VEL
LIN {X 0,Y 431.572,Z 457.85,A -85,B 0,C 180,E1 -9578.981,E2 -9578.981} C_VEL
LIN {X 0,Y 431.334,Z 462.928,A -85,B 0,C 180,E1 -9580.662,E2 -9580.662} C_VEL
LIN {X 0,Y 431.177,Z 465.722,A -85,B 0,C 180,E1 -9581.923,E2 -9581.923} C_VEL
LIN {X 0,Y 431.087,Z 467.76,A -85,B 0,C 180,E1 -9583.202,E2 -9583.202} C_VEL
LIN {X 0,Y 431.052,Z 469.048,A -85,B 0,C 180,E1 -9584.501,E2 -9584.501} C_VEL
LIN {X 0,Y 431.038,Z 469.523,A -85,B 0,C 180,E1 -9585.828,E2 -9585.828} C_VEL
LIN {X 0,Y 430.993,Z 469.172,A -85,B 0,C 180,E1 -9587.192,E2 -9587.192} C_VEL
LIN {X 0,Y 431.076,Z 467.945,A -85,B 0,C 180,E1 -9588.573,E2 -9588.573} C_VEL
LIN {X 0,Y 431.14,Z 465.743,A -85,B 0,C 180,E1 -9589.995,E2 -9589.995} C_VEL
LIN {X 0,Y 431.359,Z 461.637,A -85,B 0,C 180,E1 -9591.751,E2 -9591.751} C_VEL
LIN {X 0,Y 431.643,Z 455.652,A -85,B 0,C 180,E1 -9593.54,E2 -9593.54} C_VEL
LIN {X 0,Y 432.048,Z 448.849,A -85,B 0,C 180,E1 -9595.089,E2 -9595.089} C_VEL
LIN {X 0,Y 432.426,Z 441.281,A -85,B 0,C 180,E1 -9596.458,E2 -9596.458} C_VEL
LIN {X 0,Y 433.012,Z 432.368,A -85,B 0,C 180,E1 -9597.755,E2 -9597.755} C_VEL
LIN {X 0,Y 433.626,Z 421.875,A -85,B 0,C 180,E1 -9598.992,E2 -9598.992} C_VEL
LIN {X 0,Y 434.274,Z 411.033,A -85,B 0,C 180,E1 -9600.005,E2 -9600.005} C_VEL
LIN {X 0,Y 434.881,Z 399.701,A -85,B 0,C 180,E1 -9600.846,E2 -9600.846} C_VEL
LIN {X 0,Y 435.487,Z 386.922,A -85,B 0,C 180,E1 -9601.573,E2 -9601.573} C_VEL
LIN {X 0,Y 435.899,Z 373.949,A -85,B 0,C 180,E1 -9602.093,E2 -9602.093} C_VEL
LIN {X 0,Y 436.241,Z 360.188,A -85,B 0,C 180,E1 -9602.439,E2 -9602.439} C_VEL
LIN {X 0,Y 436.752,Z 313.421,A -85,B 0,C 180,E1 -9603.241,E2 -9603.241} C_VEL
LIN {X 0,Y 436.107,Z 307.621,A -85,B 0,C 180,E1 -9603.368,E2 -9603.368} C_VEL
LIN {X 0,Y 430.885,Z 288.936,A -85,B 0,C 180,E1 -9603.909,E2 -9603.909} C_VEL
LIN {X 0,Y 430.325,Z 283.136,A -85,B 0,C 180,E1 -9604.037,E2 -9604.037} C_VEL
LIN {X 0,Y 430.176,Z 277.835,A -85,B 0,C 180,E1 -9604.139,E2 -9604.139} C_VEL
LIN {X 0,Y 426.753,Z 258.842,A -85,B 0,C 180,E1 -9604.65,E2 -9604.65} C_VEL
LIN {X 0,Y 427.089,Z 252.655,A -85,B 0,C 180,E1 -9605.968,E2 -9605.968} C_VEL
LIN {X 0,Y 427.473,Z 246.257,A -85,B 0,C 180,E1 -9607.407,E2 -9607.407} C_VEL
LIN {X 0,Y 426.188,Z 238.64,A -85,B 0,C 180,E1 -9609.237,E2 -9609.237} C_VEL
LIN {X 0,Y 425.341,Z 234.038,A -85,B 0,C 180,E1 -9610.418,E2 -9610.418} C_VEL
LIN {X 0,Y 425.324,Z 234.002,A -85,B 0,C 180,E1 -9613.688,E2 -9613.688} C_VEL
LIN {X 0,Y 425.331,Z 234.001,A -85,B 0,C 180,E1 -9617.088,E2 -9617.088} C_VEL
LIN {X 0,Y 425.332,Z 234.004,A -85,B 0,C 180,E1 -9620.491,E2 -9620.491} C_VEL
LIN {X 0,Y 425.457,Z 233.985,A -85,B 0,C 180,E1 -9623.362,E2 -9623.362} C_VEL
LIN {X 0,Y 425.308,Z 234.005,A -85,B 0,C 180,E1 -9625.262,E2 -9625.262} C_VEL
LIN {X 0,Y 425.502,Z 233.978,A -85,B 0,C 180,E1 -9628.109,E2 -9628.109} C_VEL
LIN {X 0,Y 425.629,Z 233.962,A -85,B 0,C 180,E1 -9630.002,E2 -9630.002} C_VEL
LIN {X 0,Y 425.494,Z 233.983,A -85,B 0,C 180,E1 -9632.842,E2 -9632.842} C_VEL
LIN {X 0,Y 425.505,Z 233.979,A -85,B 0,C 180,E1 -9635.689,E2 -9635.689} C_VEL
LIN {X 0,Y 425.371,Z 233.994,A -85,B 0,C 180,E1 -9638.553,E2 -9638.553} C_VEL
LIN {X 0,Y 425.362,Z 233.995,A -85,B 0,C 180,E1 -9642.405,E2 -9642.405} C_VEL
LIN {X 0,Y 425.319,Z 234.001,A -85,B 0,C 180,E1 -9646.316,E2 -9646.316} C_VEL
LIN {X 0,Y 425.261,Z 234.016,A -85,B 0,C 180,E1 -9649.64,E2 -9649.64} C_VEL
LIN {X 0,Y 425.244,Z 234.013,A -85,B 0,C 180,E1 -9653.37,E2 -9653.37} C_VEL
LIN {X 0,Y 425.288,Z 234.004,A -85,B 0,C 180,E1 -9656.85,E2 -9656.85} C_VEL
LIN {X 0,Y 425.26,Z 234.012,A -85,B 0,C 180,E1 -9659.723,E2 -9659.723} C_VEL
LIN {X 0,Y 425.229,Z 234.012,A -85,B 0,C 180,E1 -9663.054,E2 -9663.054} C_VEL
LIN {X 0,Y 425.232,Z 234.016,A -85,B 0,C 180,E1 -9665.935,E2 -9665.935} C_VEL
LIN {X 0,Y 425.261,Z 234.008,A -85,B 0,C 180,E1 -9669.052,E2 -9669.052} C_VEL
LIN {X 0,Y 425.287,Z 234.01,A -85,B 0,C 180,E1 -9672.653,E2 -9672.653} C_VEL
LIN {X 0,Y 425.294,Z 234.006,A -85,B 0,C 180,E1 -9676.061,E2 -9676.061} C_VEL
LIN {X 0,Y 425.272,Z 234.014,A -85,B 0,C 180,E1 -9678.633,E2 -9678.633} C_VEL
LIN {X 0,Y 425.288,Z 234.008,A -85,B 0,C 180,E1 -9681.111,E2 -9681.111} C_VEL
LIN {X 0,Y 425.268,Z 234.012,A -85,B 0,C 180,E1 -9684.672,E2 -9684.672} C_VEL
LIN {X 0,Y 425.236,Z 234.011,A -85,B 0,C 180,E1 -9688.081,E2 -9688.081} C_VEL
LIN {X 0,Y 425.308,Z 234.006,A -85,B 0,C 180,E1 -9691.375,E2 -9691.375} C_VEL
LIN {X 0,Y 425.333,Z 234.002,A -85,B 0,C 180,E1 -9693.513,E2 -9693.513} C_VEL
LIN {X 0,Y 425.269,Z 234.008,A -85,B 0,C 180,E1 -9696.641,E2 -9696.641} C_VEL
LIN {X 0,Y 425.281,Z 234.009,A -85,B 0,C 180,E1 -9699.702,E2 -9699.702} C_VEL
LIN {X 0,Y 425.323,Z 234,A -85,B 0,C 180,E1 -9702.704,E2 -9702.704} C_VEL
LIN {X 0,Y 425.34,Z 234.005,A -85,B 0,C 180,E1 -9705.657,E2 -9705.657} C_VEL
LIN {X 0,Y 425.344,Z 233.997,A -85,B 0,C 180,E1 -9708.571,E2 -9708.571} C_VEL
LIN {X 0,Y 425.406,Z 233.993,A -85,B 0,C 180,E1 -9711.456,E2 -9711.456} C_VEL
LIN {X 0,Y 425.531,Z 233.976,A -85,B 0,C 180,E1 -9714.32,E2 -9714.32} C_VEL
LIN {X 0,Y 425.574,Z 233.975,A -85,B 0,C 180,E1 -9718.114,E2 -9718.114} C_VEL
LIN {X 0,Y 425.506,Z 233.977,A -85,B 0,C 180,E1 -9720.953,E2 -9720.953} C_VEL
LIN {X 0,Y 425.52,Z 233.976,A -85,B 0,C 180,E1 -9722.846,E2 -9722.846} C_VEL
LIN {X 0,Y 425.537,Z 233.975,A -85,B 0,C 180,E1 -9725.693,E2 -9725.693} C_VEL
LIN {X 0,Y 425.407,Z 233.995,A -85,B 0,C 180,E1 -9728.556,E2 -9728.556} C_VEL
LIN {X 0,Y 425.426,Z 233.994,A -85,B 0,C 180,E1 -9732.407,E2 -9732.407} C_VEL
LIN {X 0,Y 425.404,Z 233.994,A -85,B 0,C 180,E1 -9736.316,E2 -9736.316} C_VEL
LIN {X 0,Y 425.346,Z 233.997,A -85,B 0,C 180,E1 -9739.639,E2 -9739.639} C_VEL
LIN {X 0,Y 425.306,Z 234.004,A -85,B 0,C 180,E1 -9742.343,E2 -9742.343} C_VEL
LIN {X 0,Y 425.28,Z 234.007,A -85,B 0,C 180,E1 -9745.451,E2 -9745.451} C_VEL
LIN {X 0,Y 425.32,Z 234.006,A -85,B 0,C 180,E1 -9748.862,E2 -9748.862} C_VEL
LIN {X 0,Y 425.281,Z 234.006,A -85,B 0,C 180,E1 -9751.93,E2 -9751.93} C_VEL
LIN {X 0,Y 425.315,Z 234.008,A -85,B 0,C 180,E1 -9755.339,E2 -9755.339} C_VEL
LIN {X 0,Y 425.302,Z 234.005,A -85,B 0,C 180,E1 -9758.903,E2 -9758.903} C_VEL
LIN {X 0,Y 425.265,Z 234.01,A -85,B 0,C 180,E1 -9761.953,E2 -9761.953} C_VEL
LIN {X 0,Y 425.3,Z 234.007,A -85,B 0,C 180,E1 -9765.286,E2 -9765.286} C_VEL
LIN {X 0,Y 425.268,Z 234.007,A -85,B 0,C 180,E1 -9768.619,E2 -9768.619} C_VEL
LIN {X 0,Y 425.297,Z 234.004,A -85,B 0,C 180,E1 -9771.1,E2 -9771.1} C_VEL
LIN {X 0,Y 425.316,Z 234.001,A -85,B 0,C 180,E1 -9774.664,E2 -9774.664} C_VEL
LIN {X 0,Y 425.283,Z 234.013,A -85,B 0,C 180,E1 -9778.073,E2 -9778.073} C_VEL
LIN {X 0,Y 425.33,Z 234.004,A -85,B 0,C 180,E1 -9781.366,E2 -9781.366} C_VEL
LIN {X 0,Y 425.355,Z 234.128,A -85,B 0,C 180,E1 -9783.768,E2 -9783.768} C_VEL
LIN {X 0,Y 427.668,Z 246.107,A -85,B 0,C 180,E1 -9786.514,E2 -9786.514} C_VEL
LIN {X 0,Y 427.881,Z 249.893,A -85,B 0,C 180,E1 -9787.326,E2 -9787.326} C_VEL
LIN {X 0,Y 426.736,Z 267.9,A -85,B 0,C 180,E1 -9791.042,E2 -9791.042} C_VEL
LIN {X 0,Y 426.645,Z 269.916,A -85,B 0,C 180,E1 -9791.382,E2 -9791.382} C_VEL
LIN {X 0,Y 430.323,Z 293.206,A -85,B 0,C 180,E1 -9791.982,E2 -9791.982} C_VEL
LIN {X 0,Y 429.252,Z 377.43,A -85,B 0,C 180,E1 -9793.471,E2 -9793.471} C_VEL
LIN {X 0,Y 428.893,Z 390.542,A -85,B 0,C 180,E1 -9793.885,E2 -9793.885} C_VEL
LIN {X 0,Y 428.299,Z 403.227,A -85,B 0,C 180,E1 -9794.473,E2 -9794.473} C_VEL
LIN {X 0,Y 427.628,Z 415.34,A -85,B 0,C 180,E1 -9795.24,E2 -9795.24} C_VEL
LIN {X 0,Y 426.878,Z 427.705,A -85,B 0,C 180,E1 -9796.264,E2 -9796.264} C_VEL
LIN {X 0,Y 426.274,Z 438.322,A -85,B 0,C 180,E1 -9797.38,E2 -9797.38} C_VEL
LIN {X 0,Y 425.645,Z 447.471,A -85,B 0,C 180,E1 -9798.571,E2 -9798.571} C_VEL
LIN {X 0,Y 425.081,Z 456.393,A -85,B 0,C 180,E1 -9800.001,E2 -9800.001} C_VEL
LIN {X 0,Y 424.695,Z 463.537,A -85,B 0,C 180,E1 -9801.433,E2 -9801.433} C_VEL
LIN {X 0,Y 424.378,Z 469.226,A -85,B 0,C 180,E1 -9802.864,E2 -9802.864} C_VEL
LIN {X 0,Y 424.22,Z 473.697,A -85,B 0,C 180,E1 -9804.294,E2 -9804.294} C_VEL
LIN {X 0,Y 424.213,Z 476.055,A -85,B 0,C 180,E1 -9805.247,E2 -9805.247} C_VEL
LIN {X 0,Y 424.088,Z 477.977,A -85,B 0,C 180,E1 -9806.198,E2 -9806.198} C_VEL
LIN {X 0,Y 424.092,Z 479.45,A -85,B 0,C 180,E1 -9807.149,E2 -9807.149} C_VEL
LIN {X 0,Y 424.128,Z 480.485,A -85,B 0,C 180,E1 -9808.099,E2 -9808.099} C_VEL
LIN {X 0,Y 424.068,Z 481.374,A -85,B 0,C 180,E1 -9809.998,E2 -9809.998} C_VEL
LIN {X 0,Y 424.075,Z 481.198,A -85,B 0,C 180,E1 -9810.948,E2 -9810.948} C_VEL
LIN {X 0,Y 424.128,Z 480.604,A -85,B 0,C 180,E1 -9811.898,E2 -9811.898} C_VEL
LIN {X 0,Y 424.091,Z 479.617,A -85,B 0,C 180,E1 -9812.848,E2 -9812.848} C_VEL
LIN {X 0,Y 424.087,Z 478.231,A -85,B 0,C 180,E1 -9813.799,E2 -9813.799} C_VEL
LIN {X 0,Y 424.249,Z 475.3,A -85,B 0,C 180,E1 -9815.226,E2 -9815.226} C_VEL
LIN {X 0,Y 424.319,Z 471.326,A -85,B 0,C 180,E1 -9816.656,E2 -9816.656} C_VEL
LIN {X 0,Y 424.649,Z 465.215,A -85,B 0,C 180,E1 -9818.325,E2 -9818.325} C_VEL
LIN {X 0,Y 425.044,Z 458.529,A -85,B 0,C 180,E1 -9819.756,E2 -9819.756} C_VEL
LIN {X 0,Y 425.571,Z 450.234,A -85,B 0,C 180,E1 -9821.187,E2 -9821.187} C_VEL
LIN {X 0,Y 426.24,Z 441.742,A -85,B 0,C 180,E1 -9822.375,E2 -9822.375} C_VEL
LIN {X 0,Y 426.935,Z 432.18,A -85,B 0,C 180,E1 -9823.47,E2 -9823.47} C_VEL
LIN {X 0,Y 427.552,Z 420.895,A -85,B 0,C 180,E1 -9824.516,E2 -9824.516} C_VEL
LIN {X 0,Y 428.259,Z 409.563,A -85,B 0,C 180,E1 -9825.343,E2 -9825.343} C_VEL
LIN {X 0,Y 428.927,Z 398.003,A -85,B 0,C 180,E1 -9825.988,E2 -9825.988} C_VEL
LIN {X 0,Y 429.448,Z 384.816,A -85,B 0,C 180,E1 -9826.518,E2 -9826.518} C_VEL
LIN {X 0,Y 429.835,Z 372.198,A -85,B 0,C 180,E1 -9826.839,E2 -9826.839} C_VEL
LIN {X 0,Y 430.788,Z 292.018,A -85,B 0,C 180,E1 -9828.268,E2 -9828.268} C_VEL
LIN {X 0,Y 426.849,Z 269.078,A -85,B 0,C 180,E1 -9828.922,E2 -9828.922} C_VEL
LIN {X 0,Y 427.905,Z 250.307,A -85,B 0,C 180,E1 -9832.667,E2 -9832.667} C_VEL
LIN {X 0,Y 427.783,Z 246.419,A -85,B 0,C 180,E1 -9833.476,E2 -9833.476} C_VEL
LIN {X 0,Y 425.629,Z 235.318,A -85,B 0,C 180,E1 -9835.947,E2 -9835.947} C_VEL
LIN {X 0,Y 425.33,Z 234.034,A -85,B 0,C 180,E1 -9836.329,E2 -9836.329} C_VEL
LIN {X 0,Y 425.338,Z 234.002,A -85,B 0,C 180,E1 -9838.862,E2 -9838.862} C_VEL
LIN {X 0,Y 425.273,Z 234.014,A -85,B 0,C 180,E1 -9841.924,E2 -9841.924} C_VEL
LIN {X 0,Y 425.306,Z 234.007,A -85,B 0,C 180,E1 -9845.333,E2 -9845.333} C_VEL
LIN {X 0,Y 425.286,Z 234.007,A -85,B 0,C 180,E1 -9848.897,E2 -9848.897} C_VEL
LIN {X 0,Y 425.262,Z 234.01,A -85,B 0,C 180,E1 -9852.652,E2 -9852.652} C_VEL
LIN {X 0,Y 425.288,Z 234.005,A -85,B 0,C 180,E1 -9855.279,E2 -9855.279} C_VEL
LIN {X 0,Y 425.251,Z 234.015,A -85,B 0,C 180,E1 -9858.614,E2 -9858.614} C_VEL
LIN {X 0,Y 425.278,Z 234.007,A -85,B 0,C 180,E1 -9861.094,E2 -9861.094} C_VEL
LIN {X 0,Y 425.293,Z 234.011,A -85,B 0,C 180,E1 -9864.659,E2 -9864.659} C_VEL
LIN {X 0,Y 425.262,Z 234.01,A -85,B 0,C 180,E1 -9868.068,E2 -9868.068} C_VEL
LIN {X 0,Y 425.295,Z 234.006,A -85,B 0,C 180,E1 -9871.36,E2 -9871.36} C_VEL
LIN {X 0,Y 425.255,Z 234.011,A -85,B 0,C 180,E1 -9874.547,E2 -9874.547} C_VEL
LIN {X 0,Y 425.286,Z 234.003,A -85,B 0,C 180,E1 -9877.725,E2 -9877.725} C_VEL
LIN {X 0,Y 425.318,Z 234.003,A -85,B 0,C 180,E1 -9880.697,E2 -9880.697} C_VEL
LIN {X 0,Y 425.311,Z 234.001,A -85,B 0,C 180,E1 -9883.68,E2 -9883.68} C_VEL
LIN {X 0,Y 425.384,Z 233.995,A -85,B 0,C 180,E1 -9887.091,E2 -9887.091} C_VEL
LIN {X 0,Y 425.376,Z 233.997,A -85,B 0,C 180,E1 -9890.484,E2 -9890.484} C_VEL
LIN {X 0,Y 425.489,Z 233.983,A -85,B 0,C 180,E1 -9893.355,E2 -9893.355} C_VEL
LIN {X 0,Y 425.334,Z 234.005,A -85,B 0,C 180,E1 -9895.255,E2 -9895.255} C_VEL
LIN {X 0,Y 425.549,Z 233.974,A -85,B 0,C 180,E1 -9898.101,E2 -9898.101} C_VEL
LIN {X 0,Y 425.68,Z 233.956,A -85,B 0,C 180,E1 -9899.994,E2 -9899.994} C_VEL
LIN {X 0,Y 425.525,Z 233.977,A -85,B 0,C 180,E1 -9902.834,E2 -9902.834} C_VEL
LIN {X 0,Y 425.476,Z 233.984,A -85,B 0,C 180,E1 -9906.475,E2 -9906.475} C_VEL
LIN {X 0,Y 425.378,Z 234.001,A -85,B 0,C 180,E1 -9909.503,E2 -9909.503} C_VEL
LIN {X 0,Y 425.376,Z 233.997,A -85,B 0,C 180,E1 -9912.904,E2 -9912.904} C_VEL
LIN {X 0,Y 425.33,Z 234.004,A -85,B 0,C 180,E1 -9916.599,E2 -9916.599} C_VEL
LIN {X 0,Y 425.328,Z 234.005,A -85,B 0,C 180,E1 -9919.642,E2 -9919.642} C_VEL
LIN {X 0,Y 425.347,Z 234.132,A -85,B 0,C 180,E1 -9922.174,E2 -9922.174} C_VEL
LIN {X 0,Y 427.479,Z 244.695,A -85,B 0,C 180,E1 -9924.502,E2 -9924.502} C_VEL
LIN {X 0,Y 426.969,Z 258.187,A -85,B 0,C 180,E1 -9927.134,E2 -9927.134} C_VEL
LIN {X 0,Y 430.834,Z 278.549,A -85,B 0,C 180,E1 -9927.732,E2 -9927.732} C_VEL
LIN {X 0,Y 429.716,Z 366.526,A -85,B 0,C 180,E1 -9929.324,E2 -9929.324} C_VEL
LIN {X 0,Y 429.245,Z 380.493,A -85,B 0,C 180,E1 -9929.778,E2 -9929.778} C_VEL
LIN {X 0,Y 428.769,Z 392.705,A -85,B 0,C 180,E1 -9930.369,E2 -9930.369} C_VEL
LIN {X 0,Y 428.096,Z 405.107,A -85,B 0,C 180,E1 -9931.184,E2 -9931.184} C_VEL
LIN {X 0,Y 427.365,Z 416.645,A -85,B 0,C 180,E1 -9932.158,E2 -9932.158} C_VEL
LIN {X 0,Y 426.663,Z 426.495,A -85,B 0,C 180,E1 -9933.199,E2 -9933.199} C_VEL
LIN {X 0,Y 426.015,Z 435.91,A -85,B 0,C 180,E1 -9934.43,E2 -9934.43} C_VEL
LIN {X 0,Y 425.474,Z 443.379,A -85,B 0,C 180,E1 -9935.617,E2 -9935.617} C_VEL
LIN {X 0,Y 424.968,Z 450.422,A -85,B 0,C 180,E1 -9936.978,E2 -9936.978} C_VEL
LIN {X 0,Y 424.588,Z 457.163,A -85,B 0,C 180,E1 -9938.62,E2 -9938.62} C_VEL
LIN {X 0,Y 424.286,Z 462.524,A -85,B 0,C 180,E1 -9940.366,E2 -9940.366} C_VEL
LIN {X 0,Y 424.092,Z 465.71,A -85,B 0,C 180,E1 -9941.781,E2 -9941.781} C_VEL
LIN {X 0,Y 423.991,Z 467.899,A -85,B 0,C 180,E1 -9943.173,E2 -9943.173} C_VEL
LIN {X 0,Y 423.951,Z 469.19,A -85,B 0,C 180,E1 -9944.538,E2 -9944.538} C_VEL
LIN {X 0,Y 423.934,Z 469.633,A -85,B 0,C 180,E1 -9945.874,E2 -9945.874} C_VEL
LIN {X 0,Y 423.896,Z 469.279,A -85,B 0,C 180,E1 -9947.178,E2 -9947.178} C_VEL
LIN {X 0,Y 423.968,Z 468.199,A -85,B 0,C 180,E1 -9948.469,E2 -9948.469} C_VEL
LIN {X 0,Y 424.026,Z 466.422,A -85,B 0,C 180,E1 -9949.732,E2 -9949.732} C_VEL
LIN {X 0,Y 424.182,Z 463.544,A -85,B 0,C 180,E1 -9951.128,E2 -9951.128} C_VEL
LIN {X 0,Y 424.37,Z 459.333,A -85,B 0,C 180,E1 -9952.633,E2 -9952.633} C_VEL
LIN {X 0,Y 424.696,Z 453.691,A -85,B 0,C 180,E1 -9954.165,E2 -9954.165} C_VEL
LIN {X 0,Y 425.144,Z 446.338,A -85,B 0,C 180,E1 -9955.728,E2 -9955.728} C_VEL
LIN {X 0,Y 425.696,Z 437.692,A -85,B 0,C 180,E1 -9957.189,E2 -9957.189} C_VEL
LIN {X 0,Y 426.235,Z 429.057,A -85,B 0,C 180,E1 -9958.366,E2 -9958.366} C_VEL
LIN {X 0,Y 426.859,Z 419.36,A -85,B 0,C 180,E1 -9959.449,E2 -9959.449} C_VEL
LIN {X 0,Y 427.545,Z 408.197,A -85,B 0,C 180,E1 -9960.455,E2 -9960.455} C_VEL
LIN {X 0,Y 428.128,Z 397.173,A -85,B 0,C 180,E1 -9961.24,E2 -9961.24} C_VEL
LIN {X 0,Y 428.712,Z 383.866,A -85,B 0,C 180,E1 -9961.95,E2 -9961.95} C_VEL
LIN {X 0,Y 429.098,Z 370.891,A -85,B 0,C 180,E1 -9962.437,E2 -9962.437} C_VEL
LIN {X 0,Y 429.431,Z 355.986,A -85,B 0,C 180,E1 -9962.761,E2 -9962.761} C_VEL
LIN {X 0,Y 430.325,Z 283.136,A -85,B 0,C 180,E1 -9964.037,E2 -9964.037} C_VEL
LIN {X 0,Y 429.581,Z 279.373,A -85,B 0,C 180,E1 -9964.135,E2 -9964.135} C_VEL
LIN {X 0,Y 427.045,Z 274.895,A -85,B 0,C 180,E1 -9964.319,E2 -9964.319} C_VEL
LIN {X 0,Y 422.448,Z 268.451,A -85,B 0,C 180,E1 -9964.627,E2 -9964.627} C_VEL
LIN {X 0,Y 420.91,Z 264.799,A -85,B 0,C 180,E1 -9964.759,E2 -9964.759} C_VEL
LIN {X 0,Y 419.848,Z 259.029,A -85,B 0,C 180,E1 -9964.944,E2 -9964.944} C_VEL
LIN {X 0,Y 419.868,Z 257.226,A -85,B 0,C 180,E1 -9965.264,E2 -9965.264} C_VEL
LIN {X 0,Y 420.479,Z 247.897,A -85,B 0,C 180,E1 -9967.394,E2 -9967.394} C_VEL
LIN {X 0,Y 419.578,Z 241.697,A -85,B 0,C 180,E1 -9968.894,E2 -9968.894} C_VEL
LIN {X 0,Y 418.299,Z 234.942,A -85,B 0,C 180,E1 -9970.622,E2 -9970.622} C_VEL
LIN {X 0,Y 418.253,Z 234.889,A -85,B 0,C 180,E1 -9974.406,E2 -9974.406} C_VEL
LIN {X 0,Y 418.298,Z 234.875,A -85,B 0,C 180,E1 -9977.386,E2 -9977.386} C_VEL
LIN {X 0,Y 418.288,Z 234.88,A -85,B 0,C 180,E1 -9980.329,E2 -9980.329} C_VEL
LIN {X 0,Y 418.42,Z 234.862,A -85,B 0,C 180,E1 -9983.25,E2 -9983.25} C_VEL
LIN {X 0,Y 418.278,Z 234.881,A -85,B 0,C 180,E1 -9985.183,E2 -9985.183} C_VEL
LIN {X 0,Y 418.472,Z 234.853,A -85,B 0,C 180,E1 -9988.077,E2 -9988.077} C_VEL
LIN {X 0,Y 418.599,Z 234.838,A -85,B 0,C 180,E1 -9990.002,E2 -9990.002} C_VEL
LIN {X 0,Y 418.447,Z 234.862,A -85,B 0,C 180,E1 -9992.89,E2 -9992.89} C_VEL
LIN {X 0,Y 418.46,Z 234.856,A -85,B 0,C 180,E1 -9995.785,E2 -9995.785} C_VEL
LIN {X 0,Y 418.33,Z 234.872,A -85,B 0,C 180,E1 -9998.698,E2 -9998.698} C_VEL
LIN {X 0,Y 418.267,Z 234.884,A -85,B 0,C 180,E1 -10001.634,E2 -10001.634} C_VEL
LIN {X 0,Y 418.241,Z 234.882,A -85,B 0,C 180,E1 -10004.601,E2 -10004.601} C_VEL
LIN {X 0,Y 418.22,Z 234.893,A -85,B 0,C 180,E1 -10007.608,E2 -10007.608} C_VEL
LIN {X 0,Y 418.183,Z 234.889,A -85,B 0,C 180,E1 -10010.668,E2 -10010.668} C_VEL
LIN {X 0,Y 418.226,Z 234.892,A -85,B 0,C 180,E1 -10013.786,E2 -10013.786} C_VEL
LIN {X 0,Y 418.251,Z 234.881,A -85,B 0,C 180,E1 -10017.076,E2 -10017.076} C_VEL
LIN {X 0,Y 418.205,Z 234.891,A -85,B 0,C 180,E1 -10020.277,E2 -10020.277} C_VEL
LIN {X 0,Y 418.195,Z 234.89,A -85,B 0,C 180,E1 -10023.683,E2 -10023.683} C_VEL
LIN {X 0,Y 418.195,Z 234.888,A -85,B 0,C 180,E1 -10027.23,E2 -10027.23} C_VEL
LIN {X 0,Y 418.216,Z 234.886,A -85,B 0,C 180,E1 -10029.687,E2 -10029.687} C_VEL
LIN {X 0,Y 418.24,Z 234.889,A -85,B 0,C 180,E1 -10032.336,E2 -10032.336} C_VEL
LIN {X 0,Y 418.233,Z 234.885,A -85,B 0,C 180,E1 -10035.121,E2 -10035.121} C_VEL
LIN {X 0,Y 418.254,Z 234.881,A -85,B 0,C 180,E1 -10037.781,E2 -10037.781} C_VEL
LIN {X 0,Y 418.231,Z 234.884,A -85,B 0,C 180,E1 -10041.567,E2 -10041.567} C_VEL
